# B&R Automation Studio project FeederLib
Automation Studio 4.10.2.37; technology packages: Acp10Arnc0 5.12.2, mapp 5.12.1, mappSafety 5.12.2, mappView 5.12.1

## Configuration Config1

CPU PC_any, AutomationRuntime C4.90, Build 4.1.2, Safety 0.0, Vc V4.72.2

### Task classes (Cpu.sw)
```
Cyclic#1 (cycle 2000 us, tolerance 200000 us):
  ReadData <- ReadData.prg
Cyclic#3 (cycle 100000 us):
  ReadTest <- ReadTest.prg
Binaries: mvLoader, udbdef, TCData, FWRules, arconfig, User, Role, iomap, asfw, ashwac, ashwd, sysconf, OpcUaMap
Libraries: sys_lib, AsBrStr, runtime, FeederLib, FileIO, standard, astime, arssl, asieccon
```

### Hardware
```
PC : PC_any v1.1.1.0 (OrderNumber=PC)
  ConfigurationID = FeederLib_Config1
  SystemTick = 2000
  IdleTaskClass = 4
  ActivateExceptionTaskClass = 1
  Cyclic1Duration = 2000
  Cyclic1Tolerance = 200000
  Cyclic2Duration = 50000
  Cyclic3Duration = 100000
  FileDevice1
  FileDeviceName1 = HardDisk
  FileDevicePath1 = D:\Users\stankevich.sl\Documents\FeederLib\Temp
  WebServerPort = 81
  ActivateOpcUa = 1
  OpcUaInformationModels_PV_Version = 1
```

## Configuration HW

CPU 5APC3100.KBU1-000, AutomationRuntime C4.90, Build 4.1.2, Safety 0.0, Vc V4.52.0

### Task classes (Cpu.sw)
```
Cyclic#1 (cycle 2000 us, tolerance 0 us):
  HWtest <- HWtest.prg
DataObjects: Acp10sys, assl1
NcDataObjects: acp10etxen <- acp10etxen.dob, gAxis01a <- gAxis01obj.gAxis01a.dob, gAxis01i <- gAxis01obj.gAxis01i.dob, gAxis02a <- gAxis02obj.gAxis02a.dob, gAxis02i <- gAxis02obj.gAxis02i.dob, acp10etxe1 <- acp10etxen.dob, gAxis02a1 <- gAxis02obj.gAxis02a.dob, gAxis02i1 <- gAxis02obj.gAxis02i.dob, gAxis01a1 <- gAxis01obj.gAxis01a.dob, gAxis01i1 <- gAxis01obj.gAxis01i.dob
Binaries: arsvcreg, udbdef, mvLoader, TCData, arflatprv, arcoal, Acp10map, acp10cfg, asnxdb1, Config_1, ashwd, ashwac, User, sysconf, asfw, arconfig, iomap, Role, Config, Settings, TCLang, Config_4, Config_2, Config_3, Config_7, Config_5, Config_6, Config_9, Config_8, asiol2, OpcUaMap, asiol1, AlarmCfg, AlarmHCfg, asnxdb2
Libraries: MpAxis, MpBase, NcGlobal, Acp10_MC, brsystem, Acp10man, sys_lib, Acp10par, runtime, FileIO, standard, astime, MpCom, AsBrStr, SfDomain, UserLib, asieccon, powerlnk, aruser, SfDomDrv, asusb, MpSfDomMgr, SfDomVis, arssl, asiodiag, astcp, dataobj, areventlog, UsAlarmLib, MpAlarmX, FeederLib
```

### Hardware
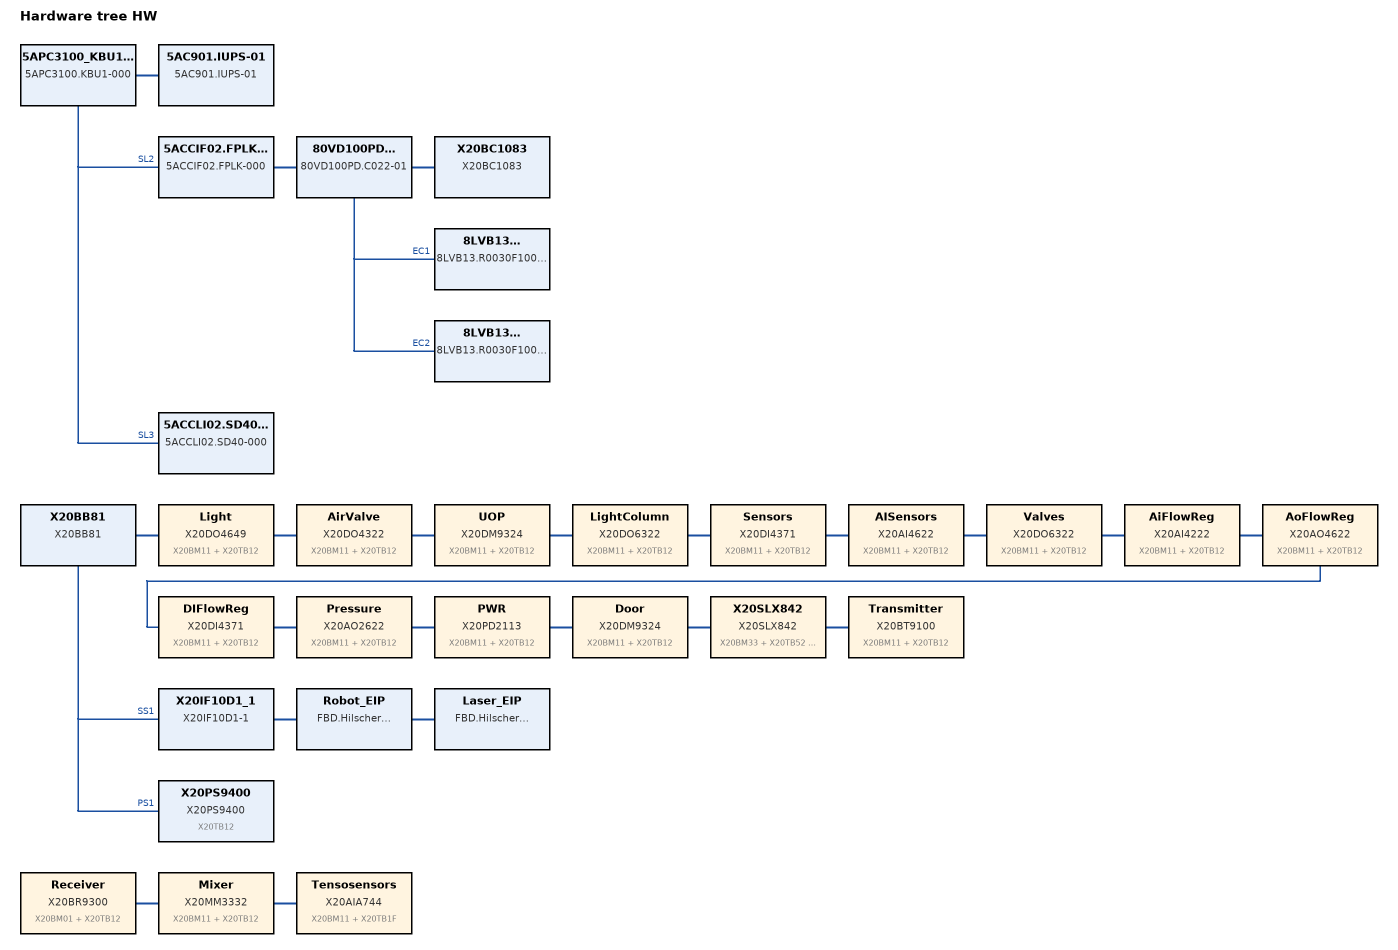
```
5AC901.IUPS-01 : 5AC901.IUPS-01 v1.3.1.0  [SL -> 5APC3100_KBU1_000.SL1]
5ACCIF02.FPLK-000 : 5ACCIF02.FPLK-000 v1.5.2.0  [SL -> 5APC3100_KBU1_000.SL2]
  Connector IF1:
    Channel1
    ChannelID1 = ACP10_MC_BROADCAST
    ChannelType1 = OCTET[24]
5ACCLI02.SD40-000 : 5ACCLI02.SD40-000 v2.0.0.0  [SL -> 5APC3100_KBU1_000.SL3]
5APC3100_KBU1_000 : 5APC3100.KBU1-000 v2.2.1.0
  Connector IF3:
    AssignedOperatingSystem = GPOS
  Connector IF4:
    AssignedOperatingSystem = ARemb
    ActivateDevice = 1
    Mode = Manual
    InternetAddress = 192.168.1.3
    SubnetMask = 255.255.255.0
  Connector IF9:
    OperatingSystem = ARemb
    ActivateDevice = 1
  Connector IF5:
    AssignedOperatingSystem = GPOS
  Connector IF6:
    AssignedOperatingSystem = GPOS
  Connector IF7:
    AssignedOperatingSystem = ARemb
  Connector IF8:
    AssignedOperatingSystem = ARemb
  ConfigurationID = 5in1
  ConfigVersion = 2.0.0
  UserPartitionSize = 100
  UserRamDevice = PCI.2.FPLK.SRAM
  UserRamSize = 520000
  RemMemDevice = PCI.2.FPLK.SRAM
  RemMemSize = 100000
  PermanentPvSize = 50
  RemanentGlobalPvSize = 1200
  EnableUsbRemoteInstall = 1
  EnableCfRemoteInstall = 1
  RebootReset = 1
  TimerDeviceType = EPLX2X
  TimerDevice = 5ACCIF02.FPLK-000.IF1
  TaskClassIdleTime = 2000
  Cyclic1Duration = 2000
  Cyclic1Tolerance = 0
  Cyclic2Tolerance = 0
  Cyclic3Tolerance = 0
  FileDevice1
  FileDeviceName1 = UserDev
  FileDevicePath1 = F:\
  FileDevice2
  FileDeviceName2 = Settings
  FileDevicePath2 = F:\Settings
  FtpUser1
  FtpUsername1 = service
  FtpUserPassword1 = FnTu9SDAOUjHE2rhZgIyHa2NFgHYN5XeFFIYZLvRcYw=
  FtpUserSalt1 = Afegl0l4
  FTPAccessRight1 = 0
  WebServerPort = 81
  ActivateOpcUa = 1
  OpcUaInformationModels_PV_Version = 1
  ActivateHypervisor = 1
80VD100PD.C022-01 : 80VD100PD.C022-01 v2.5.0.0  [PLK1 -> 5ACCIF02.FPLK-000.IF1 (NodeNumber=2) [Cable Type=PowerlinkCable, Length=10, Version=1.0.0.3]; PLK2 -> X20BC1083.PLK1 (NodeNumber=2) [Cable Type=PowerlinkCable, Length=10, Version=1.0.0.3]; EC1 -> 8LVB13.R0030F100-0.EC; EC2 -> 8LVB13.R0030F100-0a.EC; MT2 -> 8LVB13.R0030F100-0a.MT]
  MotionTP = Acp10Arnc0
  AxisIsPeriodic_r1 = on
  QuickStopIsNormallyOpen_r1 = on
  AxisIsPeriodic_r2 = on
  QuickStopIsNormallyOpen_r2 = on
8LVB13.R0030F100-0 : 8LVB13.R0030F100-0 v2.2.0.3  [EC -> 80VD100PD.C022-01.EC1; MT -> 80VD100PD.C022-01.MT1]
8LVB13.R0030F100-0a : 8LVB13.R0030F100-0 v2.2.0.3  [EC -> 80VD100PD.C022-01.EC2; MT -> 80VD100PD.C022-01.MT2]
AISensors : X20AI4622 v1.1.0.0  [SS1 -> X20TB12f.SS; SL -> X20BM11f.SL1]
  InputFilter = level 128
  ChannelType01 = 4 to 20mA
  ChannelType02 = 4 to 20mA
  ChannelType03 = 4 to 20mA
AiFlowReg : X20AI4222 v1.1.0.0  [SS1 -> X20TB12h.SS; SL -> X20BM11h.SL1]
AirValve : X20DO4322 v1.1.0.0  [SS1 -> X20TB12b.SS; SL -> X20BM11b.SL1]
AoFlowReg : X20AO4622 v1.2.0.0  [SS1 -> X20TB12j.SS; SL -> X20BM11j.SL1]
DIFlowReg : X20DI4371 v1.1.0.0  [SS1 -> X20TB12k.SS; SL -> X20BM11k.SL1]
Door : X20DM9324 v1.1.0.0  [SS1 -> X20TB12.SS; SL -> X20BM11.SL1]
Laser_EIP : FBD.Hilscher.EIGAdapterDTM.ENIP Generic Adapter v1.1100.6.6839 (OrderNumber=ENIP Generic Adapter, VendorAddress=192.168.10.1)  [EIP1 -> Robot_EIP.EIP2]
  DtmId = 5db86292-2f64-4b3a-8f97-36f326a2392b
  ChannelBlocks_1ab36399-b97a-45c0-9e04-50eb06144ae9  // Module 0
  IO_InputImage_1ab36399-b97a-45c0-9e04-50eb06144ae9  // 2 Byte(s)
  Channel_1_IO_InputImage_1ab36399-b97a-45c0-9e04-50eb06144ae9
  Name_Channel_1_IO_InputImage_1ab36399-b97a-45c0-9e04-50eb06144ae9 = Laser_is_assigned
  Channel_2_IO_InputImage_1ab36399-b97a-45c0-9e04-50eb06144ae9
  Name_Channel_2_IO_InputImage_1ab36399-b97a-45c0-9e04-50eb06144ae9 = Laser_is_ON
  Channel_3_IO_InputImage_1ab36399-b97a-45c0-9e04-50eb06144ae9
  Name_Channel_3_IO_InputImage_1ab36399-b97a-45c0-9e04-50eb06144ae9 = System_error
  Channel_4_IO_InputImage_1ab36399-b97a-45c0-9e04-50eb06144ae9
  Name_Channel_4_IO_InputImage_1ab36399-b97a-45c0-9e04-50eb06144ae9 = Guide_laser_is_ON
  Channel_5_IO_InputImage_1ab36399-b97a-45c0-9e04-50eb06144ae9
  Name_Channel_5_IO_InputImage_1ab36399-b97a-45c0-9e04-50eb06144ae9 = Program_active
  Channel_6_IO_InputImage_1ab36399-b97a-45c0-9e04-50eb06144ae9
  Name_Channel_6_IO_InputImage_1ab36399-b97a-45c0-9e04-50eb06144ae9 = End_of_program
  Channel_7_IO_InputImage_1ab36399-b97a-45c0-9e04-50eb06144ae9
  Name_Channel_7_IO_InputImage_1ab36399-b97a-45c0-9e04-50eb06144ae9 = Program_is_interrupted
  Channel_8_IO_InputImage_1ab36399-b97a-45c0-9e04-50eb06144ae9
  Name_Channel_8_IO_InputImage_1ab36399-b97a-45c0-9e04-50eb06144ae9 = Analog_control_is_ON
  Channel_9_IO_InputImage_1ab36399-b97a-45c0-9e04-50eb06144ae9
  Name_Channel_9_IO_InputImage_1ab36399-b97a-45c0-9e04-50eb06144ae9 = System_warning
  Channel_10_IO_InputImage_1ab36399-b97a-45c0-9e04-50eb06144ae9
  Name_Channel_10_IO_InputImage_1ab36399-b97a-45c0-9e04-50eb06144ae9 = Laser_is_ready
  Channel_11_IO_InputImage_1ab36399-b97a-45c0-9e04-50eb06144ae9
  Name_Channel_11_IO_InputImage_1ab36399-b97a-45c0-9e04-50eb06144ae9 = Emission_is_ON
  Channel_12_IO_InputImage_1ab36399-b97a-45c0-9e04-50eb06144ae9
  Name_Channel_12_IO_InputImage_1ab36399-b97a-45c0-9e04-50eb06144ae9 = Synchronization_output
  Channel_13_IO_InputImage_1ab36399-b97a-45c0-9e04-50eb06144ae9
  Name_Channel_13_IO_InputImage_1ab36399-b97a-45c0-9e04-50eb06144ae9 = Robot_mode
  Channel_14_IO_InputImage_1ab36399-b97a-45c0-9e04-50eb06144ae9
  Name_Channel_14_IO_InputImage_1ab36399-b97a-45c0-9e04-50eb06144ae9 = Interlock
  Channel_15_IO_InputImage_1ab36399-b97a-45c0-9e04-50eb06144ae9
  Name_Channel_15_IO_InputImage_1ab36399-b97a-45c0-9e04-50eb06144ae9 = Laser_alive
  Channel_16_IO_InputImage_1ab36399-b97a-45c0-9e04-50eb06144ae9
  Name_Channel_16_IO_InputImage_1ab36399-b97a-45c0-9e04-50eb06144ae9 = Ext_software_control_is_active
  Channel_17_IO_InputImage_1ab36399-b97a-45c0-9e04-50eb06144ae9
  Name_Channel_17_IO_InputImage_1ab36399-b97a-45c0-9e04-50eb06144ae9 = Output_power
  Type_Channel_17_IO_InputImage_1ab36399-b97a-45c0-9e04-50eb06144ae9 = UINT
  Channel_18_IO_InputImage_1ab36399-b97a-45c0-9e04-50eb06144ae9
  Name_Channel_18_IO_InputImage_1ab36399-b97a-45c0-9e04-50eb06144ae9 = Optical_channel
  Type_Channel_18_IO_InputImage_1ab36399-b97a-45c0-9e04-50eb06144ae9 = USINT
  Channel_19_IO_InputImage_1ab36399-b97a-45c0-9e04-50eb06144ae9
  Name_Channel_19_IO_InputImage_1ab36399-b97a-45c0-9e04-50eb06144ae9 = Program_number
  Type_Channel_19_IO_InputImage_1ab36399-b97a-45c0-9e04-50eb06144ae9 = USINT
  Channel_20_IO_InputImage_1ab36399-b97a-45c0-9e04-50eb06144ae9
  Name_Channel_20_IO_InputImage_1ab36399-b97a-45c0-9e04-50eb06144ae9 = Laser_error
  Channel_21_IO_InputImage_1ab36399-b97a-45c0-9e04-50eb06144ae9
  Name_Channel_21_IO_InputImage_1ab36399-b97a-45c0-9e04-50eb06144ae9 = Laser_warning
  Channel_22_IO_InputImage_1ab36399-b97a-45c0-9e04-50eb06144ae9
  Name_Channel_22_IO_InputImage_1ab36399-b97a-45c0-9e04-50eb06144ae9 = Chiller_error
  Channel_23_IO_InputImage_1ab36399-b97a-45c0-9e04-50eb06144ae9
  Name_Channel_23_IO_InputImage_1ab36399-b97a-45c0-9e04-50eb06144ae9 = Chiller_warning
  Channel_24_IO_InputImage_1ab36399-b97a-45c0-9e04-50eb06144ae9
  Name_Channel_24_IO_InputImage_1ab36399-b97a-45c0-9e04-50eb06144ae9 = Safety_open
  Channel_25_IO_InputImage_1ab36399-b97a-45c0-9e04-50eb06144ae9
  Name_Channel_25_IO_InputImage_1ab36399-b97a-45c0-9e04-50eb06144ae9 = Channel_error
  Channel_26_IO_InputImage_1ab36399-b97a-45c0-9e04-50eb06144ae9
  Name_Channel_26_IO_InputImage_1ab36399-b97a-45c0-9e04-50eb06144ae9 = Laser_is_busy
  Channel_27_IO_InputImage_1ab36399-b97a-45c0-9e04-50eb06144ae9
  Name_Channel_27_IO_InputImage_1ab36399-b97a-45c0-9e04-50eb06144ae9 = Slot_error
  Channel_28_IO_InputImage_1ab36399-b97a-45c0-9e04-50eb06144ae9
  Name_Channel_28_IO_InputImage_1ab36399-b97a-45c0-9e04-50eb06144ae9 = Cabinet_door_open
  Channel_29_IO_InputImage_1ab36399-b97a-45c0-9e04-50eb06144ae9
  Name_Channel_29_IO_InputImage_1ab36399-b97a-45c0-9e04-50eb06144ae9 = Reserved_module_is_active
  Channel_30_IO_InputImage_1ab36399-b97a-45c0-9e04-50eb06144ae9
  Name_Channel_30_IO_InputImage_1ab36399-b97a-45c0-9e04-50eb06144ae9 = Reduced_active_modules
  Channel_31_IO_InputImage_1ab36399-b97a-45c0-9e04-50eb06144ae9
  Name_Channel_31_IO_InputImage_1ab36399-b97a-45c0-9e04-50eb06144ae9 = Reserved1
  Channel_32_IO_InputImage_1ab36399-b97a-45c0-9e04-50eb06144ae9
  Name_Channel_32_IO_InputImage_1ab36399-b97a-45c0-9e04-50eb06144ae9 = Module_power_supply_warning
  Channel_33_IO_InputImage_1ab36399-b97a-45c0-9e04-50eb06144ae9
  Name_Channel_33_IO_InputImage_1ab36399-b97a-45c0-9e04-50eb06144ae9 = Reserved2
  Channel_34_IO_InputImage_1ab36399-b97a-45c0-9e04-50eb06144ae9
  Name_Channel_34_IO_InputImage_1ab36399-b97a-45c0-9e04-50eb06144ae9 = Reserved3
  Channel_35_IO_InputImage_1ab36399-b97a-45c0-9e04-50eb06144ae9
  Name_Channel_35_IO_InputImage_1ab36399-b97a-45c0-9e04-50eb06144ae9 = Reserved4
  Channel_36_IO_InputImage_1ab36399-b97a-45c0-9e04-50eb06144ae9
  Name_Channel_36_IO_InputImage_1ab36399-b97a-45c0-9e04-50eb06144ae9 = Laser_number
  Type_Channel_36_IO_InputImage_1ab36399-b97a-45c0-9e04-50eb06144ae9 = USINT
  Channel_37_IO_InputImage_1ab36399-b97a-45c0-9e04-50eb06144ae9
  Name_Channel_37_IO_InputImage_1ab36399-b97a-45c0-9e04-50eb06144ae9 = Reserver5
  Type_Channel_37_IO_InputImage_1ab36399-b97a-45c0-9e04-50eb06144ae9 = USINT
  IO_OutputImage_1ab36399-b97a-45c0-9e04-50eb06144ae9  // 2 Byte(s)
  Channel_1_IO_OutputImage_1ab36399-b97a-45c0-9e04-50eb06144ae9
  Name_Channel_1_IO_OutputImage_1ab36399-b97a-45c0-9e04-50eb06144ae9 = Laser_request
  Channel_2_IO_OutputImage_1ab36399-b97a-45c0-9e04-50eb06144ae9
  Name_Channel_2_IO_OutputImage_1ab36399-b97a-45c0-9e04-50eb06144ae9 = Laser_ON
  Channel_3_IO_OutputImage_1ab36399-b97a-45c0-9e04-50eb06144ae9
  Name_Channel_3_IO_OutputImage_1ab36399-b97a-45c0-9e04-50eb06144ae9 = Reset_errors
  Channel_4_IO_OutputImage_1ab36399-b97a-45c0-9e04-50eb06144ae9
  Name_Channel_4_IO_OutputImage_1ab36399-b97a-45c0-9e04-50eb06144ae9 = Guide_laser_ON
  Channel_5_IO_OutputImage_1ab36399-b97a-45c0-9e04-50eb06144ae9
  Name_Channel_5_IO_OutputImage_1ab36399-b97a-45c0-9e04-50eb06144ae9 = Program_start
  Channel_6_IO_OutputImage_1ab36399-b97a-45c0-9e04-50eb06144ae9
  Name_Channel_6_IO_OutputImage_1ab36399-b97a-45c0-9e04-50eb06144ae9 = Program_stop
  Channel_7_IO_OutputImage_1ab36399-b97a-45c0-9e04-50eb06144ae9
  Name_Channel_7_IO_OutputImage_1ab36399-b97a-45c0-9e04-50eb06144ae9 = Reserved7
  Channel_8_IO_OutputImage_1ab36399-b97a-45c0-9e04-50eb06144ae9
  Name_Channel_8_IO_OutputImage_1ab36399-b97a-45c0-9e04-50eb06144ae9 = Analog_control_ON
  Channel_9_IO_OutputImage_1ab36399-b97a-45c0-9e04-50eb06144ae9
  Name_Channel_9_IO_OutputImage_1ab36399-b97a-45c0-9e04-50eb06144ae9 = Enable_ext_software_control
  Channel_10_IO_OutputImage_1ab36399-b97a-45c0-9e04-50eb06144ae9
  Name_Channel_10_IO_OutputImage_1ab36399-b97a-45c0-9e04-50eb06144ae9 = Set_ramp_up
  Channel_11_IO_OutputImage_1ab36399-b97a-45c0-9e04-50eb06144ae9
  Name_Channel_11_IO_OutputImage_1ab36399-b97a-45c0-9e04-50eb06144ae9 = Set_ramp_down
  Channel_12_IO_OutputImage_1ab36399-b97a-45c0-9e04-50eb06144ae9
  Name_Channel_12_IO_OutputImage_1ab36399-b97a-45c0-9e04-50eb06144ae9 = Synchronization_input
  Channel_13_IO_OutputImage_1ab36399-b97a-45c0-9e04-50eb06144ae9
  Name_Channel_13_IO_OutputImage_1ab36399-b97a-45c0-9e04-50eb06144ae9 = Reserved8
  Channel_14_IO_OutputImage_1ab36399-b97a-45c0-9e04-50eb06144ae9
  Name_Channel_14_IO_OutputImage_1ab36399-b97a-45c0-9e04-50eb06144ae9 = Reserved9
  Channel_15_IO_OutputImage_1ab36399-b97a-45c0-9e04-50eb06144ae9
  Name_Channel_15_IO_OutputImage_1ab36399-b97a-45c0-9e04-50eb06144ae9 = Reserved10
  Channel_16_IO_OutputImage_1ab36399-b97a-45c0-9e04-50eb06144ae9
  Name_Channel_16_IO_OutputImage_1ab36399-b97a-45c0-9e04-50eb06144ae9 = External_error
  Channel_17_IO_OutputImage_1ab36399-b97a-45c0-9e04-50eb06144ae9
  Name_Channel_17_IO_OutputImage_1ab36399-b97a-45c0-9e04-50eb06144ae9 = Power
  Type_Channel_17_IO_OutputImage_1ab36399-b97a-45c0-9e04-50eb06144ae9 = UINT
  Channel_18_IO_OutputImage_1ab36399-b97a-45c0-9e04-50eb06144ae9
  Name_Channel_18_IO_OutputImage_1ab36399-b97a-45c0-9e04-50eb06144ae9 = Optical_channel_
  Type_Channel_18_IO_OutputImage_1ab36399-b97a-45c0-9e04-50eb06144ae9 = USINT
  Channel_19_IO_OutputImage_1ab36399-b97a-45c0-9e04-50eb06144ae9
  Name_Channel_19_IO_OutputImage_1ab36399-b97a-45c0-9e04-50eb06144ae9 = Program_number_
  Type_Channel_19_IO_OutputImage_1ab36399-b97a-45c0-9e04-50eb06144ae9 = USINT
  Channel_20_IO_OutputImage_1ab36399-b97a-45c0-9e04-50eb06144ae9
  Name_Channel_20_IO_OutputImage_1ab36399-b97a-45c0-9e04-50eb06144ae9 = Ramping_time
  Type_Channel_20_IO_OutputImage_1ab36399-b97a-45c0-9e04-50eb06144ae9 = UINT
  Channel_21_IO_OutputImage_1ab36399-b97a-45c0-9e04-50eb06144ae9
  Name_Channel_21_IO_OutputImage_1ab36399-b97a-45c0-9e04-50eb06144ae9 = Laser_number_
  Type_Channel_21_IO_OutputImage_1ab36399-b97a-45c0-9e04-50eb06144ae9 = USINT
  Channel_22_IO_OutputImage_1ab36399-b97a-45c0-9e04-50eb06144ae9
  Name_Channel_22_IO_OutputImage_1ab36399-b97a-45c0-9e04-50eb06144ae9 = Reserved6
  Type_Channel_22_IO_OutputImage_1ab36399-b97a-45c0-9e04-50eb06144ae9 = USINT
Light : X20DO4649 v1.1.0.0  [SS1 -> X20TB12a.SS; SL -> X20BM11a.SL1]
LightColumn : X20DO6322 v1.1.0.0  [SS1 -> X20TB12d.SS; SL -> X20BM11d.SL1]
Mixer : X20MM3332 v1.1.0.0  [SS1 -> X20TB12p.SS; SL -> X20BM11o.SL1]
PWR : X20PD2113 v1.1.0.0  [SS1 -> X20TB12m.SS; SL -> X20BM11m.SL1]
Pressure : X20AO2622 v1.2.0.0  [SS1 -> X20TB12l.SS; SL -> X20BM11l.SL1]
Receiver : X20BR9300 v1.1.0.0  [SS1 -> X20TB12o.SS; SL -> X20BM01a.SL1; X2X1 -> Transmitter.X2X1 [Cable Type=X2XCable, Length=10, Version=1.0.0.3]]
Robot_EIP : FBD.Hilscher.EIGAdapterDTM.ENIP Generic Adapter v1.1100.6.6839 (OrderNumber=ENIP Generic Adapter, VendorAddress=192.168.10.2)  [EIP1 -> X20IF10D1_1.IF1]
  DtmId = aba9a34a-c52a-40cf-8487-2c047c18b069
  ChannelBlocks_9f1ee490-7d39-4fa2-ab93-255e4565e3a3  // Module 0
  IO_InputImage_9f1ee490-7d39-4fa2-ab93-255e4565e3a3  // 2 Byte(s)
  Channel_1_IO_InputImage_9f1ee490-7d39-4fa2-ab93-255e4565e3a3
  Name_Channel_1_IO_InputImage_9f1ee490-7d39-4fa2-ab93-255e4565e3a3 = Robot_DO_1
  Channel_2_IO_InputImage_9f1ee490-7d39-4fa2-ab93-255e4565e3a3
  Name_Channel_2_IO_InputImage_9f1ee490-7d39-4fa2-ab93-255e4565e3a3 = Robot_DO_2
  Channel_3_IO_InputImage_9f1ee490-7d39-4fa2-ab93-255e4565e3a3
  Name_Channel_3_IO_InputImage_9f1ee490-7d39-4fa2-ab93-255e4565e3a3 = Robot_DO_3
  Channel_4_IO_InputImage_9f1ee490-7d39-4fa2-ab93-255e4565e3a3
  Name_Channel_4_IO_InputImage_9f1ee490-7d39-4fa2-ab93-255e4565e3a3 = Robot_DO_4
  Channel_5_IO_InputImage_9f1ee490-7d39-4fa2-ab93-255e4565e3a3
  Name_Channel_5_IO_InputImage_9f1ee490-7d39-4fa2-ab93-255e4565e3a3 = Robot_DO_5
  Channel_6_IO_InputImage_9f1ee490-7d39-4fa2-ab93-255e4565e3a3
  Name_Channel_6_IO_InputImage_9f1ee490-7d39-4fa2-ab93-255e4565e3a3 = Robot_DO_6
  Channel_7_IO_InputImage_9f1ee490-7d39-4fa2-ab93-255e4565e3a3
  Name_Channel_7_IO_InputImage_9f1ee490-7d39-4fa2-ab93-255e4565e3a3 = Robot_DO_7
  Channel_8_IO_InputImage_9f1ee490-7d39-4fa2-ab93-255e4565e3a3
  Name_Channel_8_IO_InputImage_9f1ee490-7d39-4fa2-ab93-255e4565e3a3 = Robot_DO_8
  Channel_9_IO_InputImage_9f1ee490-7d39-4fa2-ab93-255e4565e3a3
  Name_Channel_9_IO_InputImage_9f1ee490-7d39-4fa2-ab93-255e4565e3a3 = Robot_DO_9
  Channel_10_IO_InputImage_9f1ee490-7d39-4fa2-ab93-255e4565e3a3
  Name_Channel_10_IO_InputImage_9f1ee490-7d39-4fa2-ab93-255e4565e3a3 = Robot_DO_10
  Channel_11_IO_InputImage_9f1ee490-7d39-4fa2-ab93-255e4565e3a3
  Name_Channel_11_IO_InputImage_9f1ee490-7d39-4fa2-ab93-255e4565e3a3 = Robot_DO_11
  Channel_12_IO_InputImage_9f1ee490-7d39-4fa2-ab93-255e4565e3a3
  Name_Channel_12_IO_InputImage_9f1ee490-7d39-4fa2-ab93-255e4565e3a3 = Robot_DO_12
  Channel_13_IO_InputImage_9f1ee490-7d39-4fa2-ab93-255e4565e3a3
  Name_Channel_13_IO_InputImage_9f1ee490-7d39-4fa2-ab93-255e4565e3a3 = Robot_DO_13
  Channel_14_IO_InputImage_9f1ee490-7d39-4fa2-ab93-255e4565e3a3
  Name_Channel_14_IO_InputImage_9f1ee490-7d39-4fa2-ab93-255e4565e3a3 = Robot_DO_14
  Channel_15_IO_InputImage_9f1ee490-7d39-4fa2-ab93-255e4565e3a3
  Name_Channel_15_IO_InputImage_9f1ee490-7d39-4fa2-ab93-255e4565e3a3 = Robot_DO_15
  Channel_16_IO_InputImage_9f1ee490-7d39-4fa2-ab93-255e4565e3a3
  Name_Channel_16_IO_InputImage_9f1ee490-7d39-4fa2-ab93-255e4565e3a3 = Robot_DO_16
  Channel_17_IO_InputImage_9f1ee490-7d39-4fa2-ab93-255e4565e3a3
  Name_Channel_17_IO_InputImage_9f1ee490-7d39-4fa2-ab93-255e4565e3a3 = Robot_DO_17
  Channel_18_IO_InputImage_9f1ee490-7d39-4fa2-ab93-255e4565e3a3
  Name_Channel_18_IO_InputImage_9f1ee490-7d39-4fa2-ab93-255e4565e3a3 = Robot_DO_18
  Channel_19_IO_InputImage_9f1ee490-7d39-4fa2-ab93-255e4565e3a3
  Name_Channel_19_IO_InputImage_9f1ee490-7d39-4fa2-ab93-255e4565e3a3 = Robot_DO_19
  Channel_20_IO_InputImage_9f1ee490-7d39-4fa2-ab93-255e4565e3a3
  Name_Channel_20_IO_InputImage_9f1ee490-7d39-4fa2-ab93-255e4565e3a3 = Robot_DO_20
  Channel_21_IO_InputImage_9f1ee490-7d39-4fa2-ab93-255e4565e3a3
  Name_Channel_21_IO_InputImage_9f1ee490-7d39-4fa2-ab93-255e4565e3a3 = Robot_DO_21
  Channel_22_IO_InputImage_9f1ee490-7d39-4fa2-ab93-255e4565e3a3
  Name_Channel_22_IO_InputImage_9f1ee490-7d39-4fa2-ab93-255e4565e3a3 = Robot_DO_22
  Channel_23_IO_InputImage_9f1ee490-7d39-4fa2-ab93-255e4565e3a3
  Name_Channel_23_IO_InputImage_9f1ee490-7d39-4fa2-ab93-255e4565e3a3 = Robot_DO_23
  Channel_24_IO_InputImage_9f1ee490-7d39-4fa2-ab93-255e4565e3a3
  Name_Channel_24_IO_InputImage_9f1ee490-7d39-4fa2-ab93-255e4565e3a3 = Robot_DO_24
  Channel_25_IO_InputImage_9f1ee490-7d39-4fa2-ab93-255e4565e3a3
  Name_Channel_25_IO_InputImage_9f1ee490-7d39-4fa2-ab93-255e4565e3a3 = Robot_DO_25
  Channel_26_IO_InputImage_9f1ee490-7d39-4fa2-ab93-255e4565e3a3
  Name_Channel_26_IO_InputImage_9f1ee490-7d39-4fa2-ab93-255e4565e3a3 = Robot_DO_26
  Channel_27_IO_InputImage_9f1ee490-7d39-4fa2-ab93-255e4565e3a3
  Name_Channel_27_IO_InputImage_9f1ee490-7d39-4fa2-ab93-255e4565e3a3 = Robot_DO_27
  Channel_28_IO_InputImage_9f1ee490-7d39-4fa2-ab93-255e4565e3a3
  Name_Channel_28_IO_InputImage_9f1ee490-7d39-4fa2-ab93-255e4565e3a3 = Robot_DO_28
  Channel_29_IO_InputImage_9f1ee490-7d39-4fa2-ab93-255e4565e3a3
  Name_Channel_29_IO_InputImage_9f1ee490-7d39-4fa2-ab93-255e4565e3a3 = Robot_DO_29
  Channel_30_IO_InputImage_9f1ee490-7d39-4fa2-ab93-255e4565e3a3
  Name_Channel_30_IO_InputImage_9f1ee490-7d39-4fa2-ab93-255e4565e3a3 = Robot_DO_30
  Channel_31_IO_InputImage_9f1ee490-7d39-4fa2-ab93-255e4565e3a3
  Name_Channel_31_IO_InputImage_9f1ee490-7d39-4fa2-ab93-255e4565e3a3 = Robot_DO_31
  Channel_32_IO_InputImage_9f1ee490-7d39-4fa2-ab93-255e4565e3a3
  Name_Channel_32_IO_InputImage_9f1ee490-7d39-4fa2-ab93-255e4565e3a3 = Robot_DO_32
  Channel_33_IO_InputImage_9f1ee490-7d39-4fa2-ab93-255e4565e3a3
  Name_Channel_33_IO_InputImage_9f1ee490-7d39-4fa2-ab93-255e4565e3a3 = Robot_DO_33
  Channel_34_IO_InputImage_9f1ee490-7d39-4fa2-ab93-255e4565e3a3
  Name_Channel_34_IO_InputImage_9f1ee490-7d39-4fa2-ab93-255e4565e3a3 = Robot_DO_34
  Channel_35_IO_InputImage_9f1ee490-7d39-4fa2-ab93-255e4565e3a3
  Name_Channel_35_IO_InputImage_9f1ee490-7d39-4fa2-ab93-255e4565e3a3 = Robot_DO_35
  Channel_36_IO_InputImage_9f1ee490-7d39-4fa2-ab93-255e4565e3a3
  Name_Channel_36_IO_InputImage_9f1ee490-7d39-4fa2-ab93-255e4565e3a3 = Robot_DO_36
  Channel_37_IO_InputImage_9f1ee490-7d39-4fa2-ab93-255e4565e3a3
  Name_Channel_37_IO_InputImage_9f1ee490-7d39-4fa2-ab93-255e4565e3a3 = Robot_DO_37
  Channel_38_IO_InputImage_9f1ee490-7d39-4fa2-ab93-255e4565e3a3
  Name_Channel_38_IO_InputImage_9f1ee490-7d39-4fa2-ab93-255e4565e3a3 = Robot_DO_38
  Channel_39_IO_InputImage_9f1ee490-7d39-4fa2-ab93-255e4565e3a3
  Name_Channel_39_IO_InputImage_9f1ee490-7d39-4fa2-ab93-255e4565e3a3 = Robot_DO_39
  Channel_40_IO_InputImage_9f1ee490-7d39-4fa2-ab93-255e4565e3a3
  Name_Channel_40_IO_InputImage_9f1ee490-7d39-4fa2-ab93-255e4565e3a3 = Robot_DO_40
  Channel_41_IO_InputImage_9f1ee490-7d39-4fa2-ab93-255e4565e3a3
  Name_Channel_41_IO_InputImage_9f1ee490-7d39-4fa2-ab93-255e4565e3a3 = Robot_DO_41
  Channel_42_IO_InputImage_9f1ee490-7d39-4fa2-ab93-255e4565e3a3
  Name_Channel_42_IO_InputImage_9f1ee490-7d39-4fa2-ab93-255e4565e3a3 = Robot_DO_42
  Channel_43_IO_InputImage_9f1ee490-7d39-4fa2-ab93-255e4565e3a3
  Name_Channel_43_IO_InputImage_9f1ee490-7d39-4fa2-ab93-255e4565e3a3 = Robot_DO_43
  Channel_44_IO_InputImage_9f1ee490-7d39-4fa2-ab93-255e4565e3a3
  Name_Channel_44_IO_InputImage_9f1ee490-7d39-4fa2-ab93-255e4565e3a3 = Robot_DO_44
  Channel_45_IO_InputImage_9f1ee490-7d39-4fa2-ab93-255e4565e3a3
  Name_Channel_45_IO_InputImage_9f1ee490-7d39-4fa2-ab93-255e4565e3a3 = Robot_DO_45
  Channel_46_IO_InputImage_9f1ee490-7d39-4fa2-ab93-255e4565e3a3
  Name_Channel_46_IO_InputImage_9f1ee490-7d39-4fa2-ab93-255e4565e3a3 = Robot_DO_46
  Channel_47_IO_InputImage_9f1ee490-7d39-4fa2-ab93-255e4565e3a3
  Name_Channel_47_IO_InputImage_9f1ee490-7d39-4fa2-ab93-255e4565e3a3 = Robot_DO_47
  Channel_48_IO_InputImage_9f1ee490-7d39-4fa2-ab93-255e4565e3a3
  Name_Channel_48_IO_InputImage_9f1ee490-7d39-4fa2-ab93-255e4565e3a3 = Robot_DO_48
  Channel_49_IO_InputImage_9f1ee490-7d39-4fa2-ab93-255e4565e3a3
  Name_Channel_49_IO_InputImage_9f1ee490-7d39-4fa2-ab93-255e4565e3a3 = Robot_DO_49
  Channel_50_IO_InputImage_9f1ee490-7d39-4fa2-ab93-255e4565e3a3
  Name_Channel_50_IO_InputImage_9f1ee490-7d39-4fa2-ab93-255e4565e3a3 = Robot_DO_50
  Channel_51_IO_InputImage_9f1ee490-7d39-4fa2-ab93-255e4565e3a3
  Name_Channel_51_IO_InputImage_9f1ee490-7d39-4fa2-ab93-255e4565e3a3 = Robot_DO_51
  Channel_52_IO_InputImage_9f1ee490-7d39-4fa2-ab93-255e4565e3a3
  Name_Channel_52_IO_InputImage_9f1ee490-7d39-4fa2-ab93-255e4565e3a3 = Robot_DO_52
  Channel_53_IO_InputImage_9f1ee490-7d39-4fa2-ab93-255e4565e3a3
  Name_Channel_53_IO_InputImage_9f1ee490-7d39-4fa2-ab93-255e4565e3a3 = Robot_DO_53
  Channel_54_IO_InputImage_9f1ee490-7d39-4fa2-ab93-255e4565e3a3
  Name_Channel_54_IO_InputImage_9f1ee490-7d39-4fa2-ab93-255e4565e3a3 = Robot_DO_54
  Channel_55_IO_InputImage_9f1ee490-7d39-4fa2-ab93-255e4565e3a3
  Name_Channel_55_IO_InputImage_9f1ee490-7d39-4fa2-ab93-255e4565e3a3 = Robot_DO_55
  Channel_56_IO_InputImage_9f1ee490-7d39-4fa2-ab93-255e4565e3a3
  Name_Channel_56_IO_InputImage_9f1ee490-7d39-4fa2-ab93-255e4565e3a3 = Robot_DO_56
  Channel_57_IO_InputImage_9f1ee490-7d39-4fa2-ab93-255e4565e3a3
  Name_Channel_57_IO_InputImage_9f1ee490-7d39-4fa2-ab93-255e4565e3a3 = Robot_DO_57
  Channel_58_IO_InputImage_9f1ee490-7d39-4fa2-ab93-255e4565e3a3
  Name_Channel_58_IO_InputImage_9f1ee490-7d39-4fa2-ab93-255e4565e3a3 = Robot_DO_58
  Channel_59_IO_InputImage_9f1ee490-7d39-4fa2-ab93-255e4565e3a3
  Name_Channel_59_IO_InputImage_9f1ee490-7d39-4fa2-ab93-255e4565e3a3 = Robot_DO_59
  Channel_60_IO_InputImage_9f1ee490-7d39-4fa2-ab93-255e4565e3a3
  Name_Channel_60_IO_InputImage_9f1ee490-7d39-4fa2-ab93-255e4565e3a3 = Robot_DO_60
  Channel_61_IO_InputImage_9f1ee490-7d39-4fa2-ab93-255e4565e3a3
  Name_Channel_61_IO_InputImage_9f1ee490-7d39-4fa2-ab93-255e4565e3a3 = Robot_DO_61
  Channel_62_IO_InputImage_9f1ee490-7d39-4fa2-ab93-255e4565e3a3
  Name_Channel_62_IO_InputImage_9f1ee490-7d39-4fa2-ab93-255e4565e3a3 = Robot_DO_62
  Channel_63_IO_InputImage_9f1ee490-7d39-4fa2-ab93-255e4565e3a3
  Name_Channel_63_IO_InputImage_9f1ee490-7d39-4fa2-ab93-255e4565e3a3 = Robot_DO_63
  Channel_64_IO_InputImage_9f1ee490-7d39-4fa2-ab93-255e4565e3a3
  Name_Channel_64_IO_InputImage_9f1ee490-7d39-4fa2-ab93-255e4565e3a3 = Robot_DO_64
  Channel_65_IO_InputImage_9f1ee490-7d39-4fa2-ab93-255e4565e3a3
  Name_Channel_65_IO_InputImage_9f1ee490-7d39-4fa2-ab93-255e4565e3a3 = Robot_GO_1
  Type_Channel_65_IO_InputImage_9f1ee490-7d39-4fa2-ab93-255e4565e3a3 = UINT
  Channel_66_IO_InputImage_9f1ee490-7d39-4fa2-ab93-255e4565e3a3
  Name_Channel_66_IO_InputImage_9f1ee490-7d39-4fa2-ab93-255e4565e3a3 = Robot_GO_2
  Type_Channel_66_IO_InputImage_9f1ee490-7d39-4fa2-ab93-255e4565e3a3 = UINT
  Channel_67_IO_InputImage_9f1ee490-7d39-4fa2-ab93-255e4565e3a3
  Name_Channel_67_IO_InputImage_9f1ee490-7d39-4fa2-ab93-255e4565e3a3 = Robot_GO_3
  Type_Channel_67_IO_InputImage_9f1ee490-7d39-4fa2-ab93-255e4565e3a3 = UINT
  Channel_68_IO_InputImage_9f1ee490-7d39-4fa2-ab93-255e4565e3a3
  Name_Channel_68_IO_InputImage_9f1ee490-7d39-4fa2-ab93-255e4565e3a3 = Robot_GO_4
  Type_Channel_68_IO_InputImage_9f1ee490-7d39-4fa2-ab93-255e4565e3a3 = UINT
  Channel_69_IO_InputImage_9f1ee490-7d39-4fa2-ab93-255e4565e3a3
  Name_Channel_69_IO_InputImage_9f1ee490-7d39-4fa2-ab93-255e4565e3a3 = Robot_GO_5
  Type_Channel_69_IO_InputImage_9f1ee490-7d39-4fa2-ab93-255e4565e3a3 = UINT
  Channel_70_IO_InputImage_9f1ee490-7d39-4fa2-ab93-255e4565e3a3
  Name_Channel_70_IO_InputImage_9f1ee490-7d39-4fa2-ab93-255e4565e3a3 = Robot_GO_6
  Type_Channel_70_IO_InputImage_9f1ee490-7d39-4fa2-ab93-255e4565e3a3 = UINT
  Channel_71_IO_InputImage_9f1ee490-7d39-4fa2-ab93-255e4565e3a3
  Name_Channel_71_IO_InputImage_9f1ee490-7d39-4fa2-ab93-255e4565e3a3 = Robot_GO_7
  Type_Channel_71_IO_InputImage_9f1ee490-7d39-4fa2-ab93-255e4565e3a3 = UINT
  Channel_72_IO_InputImage_9f1ee490-7d39-4fa2-ab93-255e4565e3a3
  Name_Channel_72_IO_InputImage_9f1ee490-7d39-4fa2-ab93-255e4565e3a3 = Robot_GO_8
  Type_Channel_72_IO_InputImage_9f1ee490-7d39-4fa2-ab93-255e4565e3a3 = UINT
  Channel_73_IO_InputImage_9f1ee490-7d39-4fa2-ab93-255e4565e3a3
  Name_Channel_73_IO_InputImage_9f1ee490-7d39-4fa2-ab93-255e4565e3a3 = Robot_GO_9
  Type_Channel_73_IO_InputImage_9f1ee490-7d39-4fa2-ab93-255e4565e3a3 = UINT
  Channel_74_IO_InputImage_9f1ee490-7d39-4fa2-ab93-255e4565e3a3
  Name_Channel_74_IO_InputImage_9f1ee490-7d39-4fa2-ab93-255e4565e3a3 = Robot_GO_10
  Type_Channel_74_IO_InputImage_9f1ee490-7d39-4fa2-ab93-255e4565e3a3 = UINT
  IO_OutputImage_9f1ee490-7d39-4fa2-ab93-255e4565e3a3  // 2 Byte(s)
  Channel_1_IO_OutputImage_9f1ee490-7d39-4fa2-ab93-255e4565e3a3
  Name_Channel_1_IO_OutputImage_9f1ee490-7d39-4fa2-ab93-255e4565e3a3 = Robot_DI_1
  Channel_2_IO_OutputImage_9f1ee490-7d39-4fa2-ab93-255e4565e3a3
  Name_Channel_2_IO_OutputImage_9f1ee490-7d39-4fa2-ab93-255e4565e3a3 = Robot_DI_2
  Channel_3_IO_OutputImage_9f1ee490-7d39-4fa2-ab93-255e4565e3a3
  Name_Channel_3_IO_OutputImage_9f1ee490-7d39-4fa2-ab93-255e4565e3a3 = Robot_DI_3
  Channel_4_IO_OutputImage_9f1ee490-7d39-4fa2-ab93-255e4565e3a3
  Name_Channel_4_IO_OutputImage_9f1ee490-7d39-4fa2-ab93-255e4565e3a3 = Robot_DI_4
  Channel_5_IO_OutputImage_9f1ee490-7d39-4fa2-ab93-255e4565e3a3
  Name_Channel_5_IO_OutputImage_9f1ee490-7d39-4fa2-ab93-255e4565e3a3 = Robot_DI_5
  Channel_6_IO_OutputImage_9f1ee490-7d39-4fa2-ab93-255e4565e3a3
  Name_Channel_6_IO_OutputImage_9f1ee490-7d39-4fa2-ab93-255e4565e3a3 = Robot_DI_6
  Channel_7_IO_OutputImage_9f1ee490-7d39-4fa2-ab93-255e4565e3a3
  Name_Channel_7_IO_OutputImage_9f1ee490-7d39-4fa2-ab93-255e4565e3a3 = Robot_DI_7
  Channel_8_IO_OutputImage_9f1ee490-7d39-4fa2-ab93-255e4565e3a3
  Name_Channel_8_IO_OutputImage_9f1ee490-7d39-4fa2-ab93-255e4565e3a3 = Robot_DI_8
  Channel_9_IO_OutputImage_9f1ee490-7d39-4fa2-ab93-255e4565e3a3
  Name_Channel_9_IO_OutputImage_9f1ee490-7d39-4fa2-ab93-255e4565e3a3 = Robot_DI_9
  Channel_10_IO_OutputImage_9f1ee490-7d39-4fa2-ab93-255e4565e3a3
  Name_Channel_10_IO_OutputImage_9f1ee490-7d39-4fa2-ab93-255e4565e3a3 = Robot_DI_10
  Channel_11_IO_OutputImage_9f1ee490-7d39-4fa2-ab93-255e4565e3a3
  Name_Channel_11_IO_OutputImage_9f1ee490-7d39-4fa2-ab93-255e4565e3a3 = Robot_DI_11
  Channel_12_IO_OutputImage_9f1ee490-7d39-4fa2-ab93-255e4565e3a3
  Name_Channel_12_IO_OutputImage_9f1ee490-7d39-4fa2-ab93-255e4565e3a3 = Robot_DI_12
  Channel_13_IO_OutputImage_9f1ee490-7d39-4fa2-ab93-255e4565e3a3
  Name_Channel_13_IO_OutputImage_9f1ee490-7d39-4fa2-ab93-255e4565e3a3 = Robot_DI_13
  Channel_14_IO_OutputImage_9f1ee490-7d39-4fa2-ab93-255e4565e3a3
  Name_Channel_14_IO_OutputImage_9f1ee490-7d39-4fa2-ab93-255e4565e3a3 = Robot_DI_14
  Channel_15_IO_OutputImage_9f1ee490-7d39-4fa2-ab93-255e4565e3a3
  Name_Channel_15_IO_OutputImage_9f1ee490-7d39-4fa2-ab93-255e4565e3a3 = Robot_DI_15
  Channel_16_IO_OutputImage_9f1ee490-7d39-4fa2-ab93-255e4565e3a3
  Name_Channel_16_IO_OutputImage_9f1ee490-7d39-4fa2-ab93-255e4565e3a3 = Robot_DI_16
  Channel_17_IO_OutputImage_9f1ee490-7d39-4fa2-ab93-255e4565e3a3
  Name_Channel_17_IO_OutputImage_9f1ee490-7d39-4fa2-ab93-255e4565e3a3 = Robot_DI_17
  Channel_18_IO_OutputImage_9f1ee490-7d39-4fa2-ab93-255e4565e3a3
  Name_Channel_18_IO_OutputImage_9f1ee490-7d39-4fa2-ab93-255e4565e3a3 = Robot_DI_18
  Channel_19_IO_OutputImage_9f1ee490-7d39-4fa2-ab93-255e4565e3a3
  Name_Channel_19_IO_OutputImage_9f1ee490-7d39-4fa2-ab93-255e4565e3a3 = Robot_DI_19
  Channel_20_IO_OutputImage_9f1ee490-7d39-4fa2-ab93-255e4565e3a3
  Name_Channel_20_IO_OutputImage_9f1ee490-7d39-4fa2-ab93-255e4565e3a3 = Robot_DI_20
  Channel_21_IO_OutputImage_9f1ee490-7d39-4fa2-ab93-255e4565e3a3
  Name_Channel_21_IO_OutputImage_9f1ee490-7d39-4fa2-ab93-255e4565e3a3 = Robot_DI_21
  Channel_22_IO_OutputImage_9f1ee490-7d39-4fa2-ab93-255e4565e3a3
  Name_Channel_22_IO_OutputImage_9f1ee490-7d39-4fa2-ab93-255e4565e3a3 = Robot_DI_22
  Channel_23_IO_OutputImage_9f1ee490-7d39-4fa2-ab93-255e4565e3a3
  Name_Channel_23_IO_OutputImage_9f1ee490-7d39-4fa2-ab93-255e4565e3a3 = Robot_DI_23
  Channel_24_IO_OutputImage_9f1ee490-7d39-4fa2-ab93-255e4565e3a3
  Name_Channel_24_IO_OutputImage_9f1ee490-7d39-4fa2-ab93-255e4565e3a3 = Robot_DI_24
  Channel_25_IO_OutputImage_9f1ee490-7d39-4fa2-ab93-255e4565e3a3
  Name_Channel_25_IO_OutputImage_9f1ee490-7d39-4fa2-ab93-255e4565e3a3 = Robot_DI_25
  Channel_26_IO_OutputImage_9f1ee490-7d39-4fa2-ab93-255e4565e3a3
  Name_Channel_26_IO_OutputImage_9f1ee490-7d39-4fa2-ab93-255e4565e3a3 = Robot_DI_26
  Channel_27_IO_OutputImage_9f1ee490-7d39-4fa2-ab93-255e4565e3a3
  Name_Channel_27_IO_OutputImage_9f1ee490-7d39-4fa2-ab93-255e4565e3a3 = Robot_DI_27
  Channel_28_IO_OutputImage_9f1ee490-7d39-4fa2-ab93-255e4565e3a3
  Name_Channel_28_IO_OutputImage_9f1ee490-7d39-4fa2-ab93-255e4565e3a3 = Robot_DI_28
  Channel_29_IO_OutputImage_9f1ee490-7d39-4fa2-ab93-255e4565e3a3
  Name_Channel_29_IO_OutputImage_9f1ee490-7d39-4fa2-ab93-255e4565e3a3 = Robot_DI_29
  Channel_30_IO_OutputImage_9f1ee490-7d39-4fa2-ab93-255e4565e3a3
  Name_Channel_30_IO_OutputImage_9f1ee490-7d39-4fa2-ab93-255e4565e3a3 = Robot_DI_30
  Channel_31_IO_OutputImage_9f1ee490-7d39-4fa2-ab93-255e4565e3a3
  Name_Channel_31_IO_OutputImage_9f1ee490-7d39-4fa2-ab93-255e4565e3a3 = Robot_DI_31
  Channel_32_IO_OutputImage_9f1ee490-7d39-4fa2-ab93-255e4565e3a3
  Name_Channel_32_IO_OutputImage_9f1ee490-7d39-4fa2-ab93-255e4565e3a3 = Robot_DI_32
  Channel_33_IO_OutputImage_9f1ee490-7d39-4fa2-ab93-255e4565e3a3
  Name_Channel_33_IO_OutputImage_9f1ee490-7d39-4fa2-ab93-255e4565e3a3 = Robot_DI_33
  Channel_34_IO_OutputImage_9f1ee490-7d39-4fa2-ab93-255e4565e3a3
  Name_Channel_34_IO_OutputImage_9f1ee490-7d39-4fa2-ab93-255e4565e3a3 = Robot_DI_34
  Channel_35_IO_OutputImage_9f1ee490-7d39-4fa2-ab93-255e4565e3a3
  Name_Channel_35_IO_OutputImage_9f1ee490-7d39-4fa2-ab93-255e4565e3a3 = Robot_DI_35
  Channel_36_IO_OutputImage_9f1ee490-7d39-4fa2-ab93-255e4565e3a3
  Name_Channel_36_IO_OutputImage_9f1ee490-7d39-4fa2-ab93-255e4565e3a3 = Robot_DI_36
  Channel_37_IO_OutputImage_9f1ee490-7d39-4fa2-ab93-255e4565e3a3
  Name_Channel_37_IO_OutputImage_9f1ee490-7d39-4fa2-ab93-255e4565e3a3 = Robot_DI_37
  Channel_38_IO_OutputImage_9f1ee490-7d39-4fa2-ab93-255e4565e3a3
  Name_Channel_38_IO_OutputImage_9f1ee490-7d39-4fa2-ab93-255e4565e3a3 = Robot_DI_38
  Channel_39_IO_OutputImage_9f1ee490-7d39-4fa2-ab93-255e4565e3a3
  Name_Channel_39_IO_OutputImage_9f1ee490-7d39-4fa2-ab93-255e4565e3a3 = Robot_DI_39
  Channel_40_IO_OutputImage_9f1ee490-7d39-4fa2-ab93-255e4565e3a3
  Name_Channel_40_IO_OutputImage_9f1ee490-7d39-4fa2-ab93-255e4565e3a3 = Robot_DI_40
  Channel_41_IO_OutputImage_9f1ee490-7d39-4fa2-ab93-255e4565e3a3
  Name_Channel_41_IO_OutputImage_9f1ee490-7d39-4fa2-ab93-255e4565e3a3 = Robot_DI_41
  Channel_42_IO_OutputImage_9f1ee490-7d39-4fa2-ab93-255e4565e3a3
  Name_Channel_42_IO_OutputImage_9f1ee490-7d39-4fa2-ab93-255e4565e3a3 = Robot_DI_42
  Channel_43_IO_OutputImage_9f1ee490-7d39-4fa2-ab93-255e4565e3a3
  Name_Channel_43_IO_OutputImage_9f1ee490-7d39-4fa2-ab93-255e4565e3a3 = Robot_DI_43
  Channel_44_IO_OutputImage_9f1ee490-7d39-4fa2-ab93-255e4565e3a3
  Name_Channel_44_IO_OutputImage_9f1ee490-7d39-4fa2-ab93-255e4565e3a3 = Robot_DI_44
  Channel_45_IO_OutputImage_9f1ee490-7d39-4fa2-ab93-255e4565e3a3
  Name_Channel_45_IO_OutputImage_9f1ee490-7d39-4fa2-ab93-255e4565e3a3 = Robot_DI_45
  Channel_46_IO_OutputImage_9f1ee490-7d39-4fa2-ab93-255e4565e3a3
  Name_Channel_46_IO_OutputImage_9f1ee490-7d39-4fa2-ab93-255e4565e3a3 = Robot_DI_46
  Channel_47_IO_OutputImage_9f1ee490-7d39-4fa2-ab93-255e4565e3a3
  Name_Channel_47_IO_OutputImage_9f1ee490-7d39-4fa2-ab93-255e4565e3a3 = Robot_DI_47
  Channel_48_IO_OutputImage_9f1ee490-7d39-4fa2-ab93-255e4565e3a3
  Name_Channel_48_IO_OutputImage_9f1ee490-7d39-4fa2-ab93-255e4565e3a3 = Robot_DI_48
  Channel_49_IO_OutputImage_9f1ee490-7d39-4fa2-ab93-255e4565e3a3
  Name_Channel_49_IO_OutputImage_9f1ee490-7d39-4fa2-ab93-255e4565e3a3 = Robot_DI_49
  Channel_50_IO_OutputImage_9f1ee490-7d39-4fa2-ab93-255e4565e3a3
  Name_Channel_50_IO_OutputImage_9f1ee490-7d39-4fa2-ab93-255e4565e3a3 = Robot_DI_50
  Channel_51_IO_OutputImage_9f1ee490-7d39-4fa2-ab93-255e4565e3a3
  Name_Channel_51_IO_OutputImage_9f1ee490-7d39-4fa2-ab93-255e4565e3a3 = Robot_DI_51
  Channel_52_IO_OutputImage_9f1ee490-7d39-4fa2-ab93-255e4565e3a3
  Name_Channel_52_IO_OutputImage_9f1ee490-7d39-4fa2-ab93-255e4565e3a3 = Robot_DI_52
  Channel_53_IO_OutputImage_9f1ee490-7d39-4fa2-ab93-255e4565e3a3
  Name_Channel_53_IO_OutputImage_9f1ee490-7d39-4fa2-ab93-255e4565e3a3 = Robot_DI_53
  Channel_54_IO_OutputImage_9f1ee490-7d39-4fa2-ab93-255e4565e3a3
  Name_Channel_54_IO_OutputImage_9f1ee490-7d39-4fa2-ab93-255e4565e3a3 = Robot_DI_54
  Channel_55_IO_OutputImage_9f1ee490-7d39-4fa2-ab93-255e4565e3a3
  Name_Channel_55_IO_OutputImage_9f1ee490-7d39-4fa2-ab93-255e4565e3a3 = Robot_DI_55
  Channel_56_IO_OutputImage_9f1ee490-7d39-4fa2-ab93-255e4565e3a3
  Name_Channel_56_IO_OutputImage_9f1ee490-7d39-4fa2-ab93-255e4565e3a3 = Robot_DI_56
  Channel_57_IO_OutputImage_9f1ee490-7d39-4fa2-ab93-255e4565e3a3
  Name_Channel_57_IO_OutputImage_9f1ee490-7d39-4fa2-ab93-255e4565e3a3 = Robot_DI_57
  Channel_58_IO_OutputImage_9f1ee490-7d39-4fa2-ab93-255e4565e3a3
  Name_Channel_58_IO_OutputImage_9f1ee490-7d39-4fa2-ab93-255e4565e3a3 = Robot_DI_58
  Channel_59_IO_OutputImage_9f1ee490-7d39-4fa2-ab93-255e4565e3a3
  Name_Channel_59_IO_OutputImage_9f1ee490-7d39-4fa2-ab93-255e4565e3a3 = Robot_DI_59
  Channel_60_IO_OutputImage_9f1ee490-7d39-4fa2-ab93-255e4565e3a3
  Name_Channel_60_IO_OutputImage_9f1ee490-7d39-4fa2-ab93-255e4565e3a3 = Robot_DI_60
  Channel_61_IO_OutputImage_9f1ee490-7d39-4fa2-ab93-255e4565e3a3
  Name_Channel_61_IO_OutputImage_9f1ee490-7d39-4fa2-ab93-255e4565e3a3 = Robot_DI_61
  Channel_62_IO_OutputImage_9f1ee490-7d39-4fa2-ab93-255e4565e3a3
  Name_Channel_62_IO_OutputImage_9f1ee490-7d39-4fa2-ab93-255e4565e3a3 = Robot_DI_62
  Channel_63_IO_OutputImage_9f1ee490-7d39-4fa2-ab93-255e4565e3a3
  Name_Channel_63_IO_OutputImage_9f1ee490-7d39-4fa2-ab93-255e4565e3a3 = Robot_DI_63
  Channel_64_IO_OutputImage_9f1ee490-7d39-4fa2-ab93-255e4565e3a3
  Name_Channel_64_IO_OutputImage_9f1ee490-7d39-4fa2-ab93-255e4565e3a3 = Robot_DI_64
  Channel_65_IO_OutputImage_9f1ee490-7d39-4fa2-ab93-255e4565e3a3
  Name_Channel_65_IO_OutputImage_9f1ee490-7d39-4fa2-ab93-255e4565e3a3 = Robot_GI_1
  Type_Channel_65_IO_OutputImage_9f1ee490-7d39-4fa2-ab93-255e4565e3a3 = UINT
  Channel_66_IO_OutputImage_9f1ee490-7d39-4fa2-ab93-255e4565e3a3
  Name_Channel_66_IO_OutputImage_9f1ee490-7d39-4fa2-ab93-255e4565e3a3 = Robot_GI_2
  Type_Channel_66_IO_OutputImage_9f1ee490-7d39-4fa2-ab93-255e4565e3a3 = UINT
  Channel_67_IO_OutputImage_9f1ee490-7d39-4fa2-ab93-255e4565e3a3
  Name_Channel_67_IO_OutputImage_9f1ee490-7d39-4fa2-ab93-255e4565e3a3 = Robot_GI_3
  Type_Channel_67_IO_OutputImage_9f1ee490-7d39-4fa2-ab93-255e4565e3a3 = UINT
  Channel_68_IO_OutputImage_9f1ee490-7d39-4fa2-ab93-255e4565e3a3
  Name_Channel_68_IO_OutputImage_9f1ee490-7d39-4fa2-ab93-255e4565e3a3 = Robot_GI_4
  Type_Channel_68_IO_OutputImage_9f1ee490-7d39-4fa2-ab93-255e4565e3a3 = UINT
Sensors : X20DI4371 v1.1.0.0  [SS1 -> X20TB12e.SS; SL -> X20BM11e.SL1]
Tensosensors : X20AIA744 v1.3.0.0  [SS1 -> X20TB1F1.SS; SL -> X20BM11p.SL1]
Transmitter : X20BT9100 v1.1.0.0  [SS1 -> X20TB12n.SS; SL -> X20BM11n.SL1]
UOP : X20DM9324 v1.1.0.0  [SS1 -> X20TB12c.SS; SL -> X20BM11c.SL1]
Valves : X20DO6322 v1.1.0.0  [SS1 -> X20TB12g.SS; SL -> X20BM11g.SL1]
X20BB81 : X20BB81 v1.0.2.0
X20BC1083 : X20BC1083 v2.12.0.0  [PLK1 -> 80VD100PD.C022-01.PLK2 (NodeNumber=3) [Cable Type=PowerlinkCable, Length=10, Version=1.0.0.3]; SL -> X20BB81.SL1]
X20BM01a : X20BM01 v2.1.0.0
X20BM11 : X20BM11 v1.0.0.1  [X2X1 -> X20BM11m.X2X2]
X20BM11a : X20BM11 v1.0.0.1  [X2X1 -> X20BB81.IF1]
X20BM11b : X20BM11 v1.0.0.1  [X2X1 -> X20BM11a.X2X2]
X20BM11c : X20BM11 v1.0.0.1  [X2X1 -> X20BM11b.X2X2]
X20BM11d : X20BM11 v1.0.0.1  [X2X1 -> X20BM11c.X2X2]
X20BM11e : X20BM11 v1.0.0.1  [X2X1 -> X20BM11d.X2X2]
X20BM11f : X20BM11 v1.0.0.1  [X2X1 -> X20BM11e.X2X2]
X20BM11g : X20BM11 v1.0.0.1  [X2X1 -> X20BM11f.X2X2]
X20BM11h : X20BM11 v1.0.0.1  [X2X1 -> X20BM11g.X2X2]
X20BM11j : X20BM11 v1.0.0.1  [X2X1 -> X20BM11h.X2X2]
X20BM11k : X20BM11 v1.0.0.1  [X2X1 -> X20BM11j.X2X2]
X20BM11l : X20BM11 v1.0.0.1  [X2X1 -> X20BM11k.X2X2]
X20BM11m : X20BM11 v1.0.0.1  [X2X1 -> X20BM11l.X2X2]
X20BM11n : X20BM11 v1.0.0.1  [X2X1 -> X20BM33.X2X2]
X20BM11o : X20BM11 v1.0.0.1  [X2X1 -> X20BM01a.X2X2]
X20BM11p : X20BM11 v1.0.0.1  [X2X1 -> X20BM11o.X2X2]
X20BM33 : X20BM33 v1.0.0.6  [X2X1 -> X20BM11.X2X2]
X20IF10D1_1 : X20IF10D1-1 v1.6.0.0  [SS -> X20BB81.SS1]
  Connector IF1:
    DtmId = 89c72c1d-13b9-4e5d-9bc0-35ee8e3ffdec
  ConfigFile = X20IF10D1_1.dtm
  ConfigModule = asnxdb1
  CycleTime = 2000
X20PS9400 : X20PS9400 v1.4.0.0  [SS1 -> X20TB12q.SS; PS -> X20BB81.PS1]
  PowerInfo = on
X20SLX842 : X20SLX842 v2.2.0.0  [SS1 -> X20TB52.SS; SS2 -> X20TB52a.SS; SL -> X20BM33.SL1]
  Supervision = off
  SafeProject = SafeLOGIC-1
  SafeDesigner = 4.4.0.0
  DigitalOutput01 = viaSafeLOGIC
  DigitalOutput02 = viaSafeLOGIC
  DigitalOutput03 = viaSafeLOGIC
  DigitalOutput04 = viaSafeLOGIC
  DigitalOutput05 = viaSafeLOGIC
  DigitalOutput06 = viaSafeLOGIC
X20TB12 : X20TB12 v1.0.0.0
X20TB12a : X20TB12 v1.0.0.0
X20TB12b : X20TB12 v1.0.0.0
X20TB12c : X20TB12 v1.0.0.0
X20TB12d : X20TB12 v1.0.0.0
X20TB12e : X20TB12 v1.0.0.0
X20TB12f : X20TB12 v1.0.0.0
X20TB12g : X20TB12 v1.0.0.0
X20TB12h : X20TB12 v1.0.0.0
X20TB12j : X20TB12 v1.0.0.0
X20TB12k : X20TB12 v1.0.0.0
X20TB12l : X20TB12 v1.0.0.0
X20TB12m : X20TB12 v1.0.0.0
X20TB12n : X20TB12 v1.0.0.0
X20TB12o : X20TB12 v1.0.0.0
X20TB12p : X20TB12 v1.0.0.0
X20TB12q : X20TB12 v1.0.0.0
X20TB1F1 : X20TB1F v1.0.0.0
X20TB52 : X20TB52 v1.0.0.2
X20TB52a : X20TB52 v1.0.0.2
```

### IoMap.iom - 5APC3100_KBU1_000/IoMap.iom
```iecst
VAR_CONFIG
	Cyclic#1.::HWtest:FeederBlock.IOout.PrimaryFeeder.doMixer AT %QX."Mixer".StartChannel01;
	Cyclic#1.::HWtest:FeederBlock.IOout.SecondaryFeeder.doMixer AT %QX."Mixer".StartChannel02;
	Cyclic#1.::HWtest:FeederBlock.IOin.PrimaryFeeder.aiWeight AT %ID."Tensosensors".AnalogInput01;
	Cyclic#1.::HWtest:FeederBlock.IOin.SecondaryFeeder.aiWeight AT %ID."Tensosensors".AnalogInput02;
	Cyclic#1.::HWtest:FeederBlock.Config.PrimaryFeeder.ControlWord AT %QW."Tensosensors".ControlPacked01;
	Cyclic#1.::HWtest:FeederBlock.Config.SecondaryFeeder.ControlWord AT %QW."Tensosensors".ControlPacked02;
	Cyclic#1.::gLaserIO.Out.doPowerSupply AT %IX."X20SLX842".BOOL001;
	Cyclic#1.gSealedChamberIO.Out.BasicChamberIOOut.doBlockDoor[0] AT %QX."X20SLX842".BOOL101;
	Cyclic#1.gSealedChamberIO.In.BasicChamberIOIn.diDoorState[0].DoorIsClosed AT %QX."X20SLX842".BOOL102;
	Cyclic#1.::HWtest:FeederBlock.IOout.PrimaryFeeder.doShutOff AT %QX."Valves".DigitalOutput01;
	Cyclic#1.::HWtest:FeederBlock.IOout.SecondaryFeeder.doShutOff AT %QX."Valves".DigitalOutput02;
	Cyclic#1.::HWtest:FeederBlock.Control.PrimaryStart AT %IX."Robot_EIP".Robot_DO_5;
	Cyclic#1.::HWtest:FeederBlock.Control.SecondaryStart AT %IX."Robot_EIP".Robot_DO_6;
	Cyclic#1.::HWtest:FeederBlock.Control.PrimaryFeeder.Handler.PowderRate AT %IW."Robot_EIP".Robot_GO_3;
	Cyclic#1.::HWtest:FeederBlock.Control.PrimaryFeeder.Handler.GasRate AT %IW."Robot_EIP".Robot_GO_4;
	Cyclic#1.::HWtest:FeederBlock.Control.SecondaryFeeder.Handler.PowderRate AT %IW."Robot_EIP".Robot_GO_5;
	Cyclic#1.::HWtest:FeederBlock.IOin.SecondaryFeeder.Handler.aiGasRate AT %IW."Robot_EIP".Robot_GO_6;
	Cyclic#1.::HWtest:FeederBlock.IOout.PrimaryFeeder.aoGasRate AT %QW."AoFlowReg".AnalogOutput02;
	Cyclic#1.::HWtest:FeederBlock.IOout.SecondaryFeeder.aoGasRate AT %QW."AoFlowReg".AnalogOutput03;
END_VAR
```

### Acp10cfg.ncc - 5APC3100_KBU1_000/Motion/Acp10cfg.ncc
```
NcConfiguration (Version=5.02.1, NcSwId=Acp10)
  ACP10CF1_typ:
    cnt_nettrc_rec_drive = 150
    bufsize_trace_upload = 1200
    tc_nc_man_task = Cyclic #1
    glob_pv_as_ncobject = Yes
    ncsys_dl_broadcast = Yes
    ncsys_dl_acp_reset = Yes
    safemc_log_err_to_ax = Yes
    network_init:
      ncsw_init_execute = Yes
      automatic_execute = No
      node_nr_warning = Yes
      net_err_before_ncact = Yes
    nettrc:
      enter_parsecrec = Yes
      enter_ncaction = Yes
      save_ring_startidx = No
    cam_prof_download:
      cam_dat_dl_parallel = No
      tc_cam_dl_parallel = Task class for NC Manager task
    plk_if[0]:
      if_name = IF3
      tc_CycDat_PLCopen = Task class for NC Manager task
      mc_broadcast_extdat = No
    plk_if[1]:
      if_name = SL2.IF1
      tc_CycDat_PLCopen = Task class for NC Manager task
      mc_broadcast_extdat = No
```

### Acp10map.ncm - 5APC3100_KBU1_000/Motion/Acp10map.ncm
```
NcMapping (NcSwId=Acp10)
  NcObject gAxis01 (ModuleId=80VD100PD.C022-01, Type=ncAXIS, Channel=1, AcoposSimulation=Off, InitParameter=gAxis01i, AcoposParameter=gAxis01a, AdditionalData=PLCopen_ModPos="1000,1" , Disabled=FALSE, ModuleDisabled=FALSE)
  NcObject gAxis02 (ModuleId=80VD100PD.C022-01, Type=ncAXIS, Channel=2, AcoposSimulation=Off, InitParameter=gAxis02i, AcoposParameter=gAxis02a, AdditionalData=PLCopen_ModPos="1000,1" , Disabled=FALSE, ModuleDisabled=FALSE)
  NcObject 80VD100PD.C022-01_ncV_AXIS1 (ModuleId=80VD100PD.C022-01, Type=ncV_AXIS, Channel=1, Disabled=TRUE, ModuleDisabled=FALSE)
  NcObject 80VD100PD.C022-01_ncV_AXIS2 (ModuleId=80VD100PD.C022-01, Type=ncV_AXIS, Channel=2, Disabled=TRUE, ModuleDisabled=FALSE)
```

### Config.mpaxisbasic - 5APC3100_KBU1_000/Motion/Config.mpaxisbasic
```
Element gLinkFeeder1 (Type=mpaxisbasic)
Element gLinkFeeder2 (Type=mpaxisbasic)
```

- Safety project (password-protected, skipped)

### Alarms.mpalarmxcore - 5APC3100_KBU1_000/mappServices/Alarms.mpalarmxcore
```
Element gAlarmXCore (Type=mpalarmxcore)
  mapp.AlarmX.Core:
    BySeverity:
      [0]:
        Severity = 1
        [0] = Reaction
          Name = ReactionWarning
      [1]:
        Severity = 5
        [0] = Reaction
          Name = ReactionWarningAlarm
      [2]:
        Severity = 9
        [0] = Reaction
          Name = ReactionAlarmStopAll
      [3]:
        Severity = 10
        [0] = Reaction
          Name = ReactionAlarmSignalAndStopAll
      [4]:
        Severity = 3
        [0] = Reaction
          Name = ReactionSignal
    Default:
      [0] = Reaction
```

## Logical view

Binary libraries used (declarations not repeated): operator, runtime, astime, AsIecCon, sys_lib, AsBrStr, FileIO, standard, MpAxis, Acp10_MC, NcGlobal, MpBase, MpCom, brsystem, Acp10man, Acp10par, SfDomain, MpAlarmX

### Global.var - Global variables
```iecst
VAR
	T : ARRAY[0..2399] OF REAL;
	Ktare : ARRAY[0..2399] OF REAL;
	V : ARRAY[0..2399] OF REAL;
	W : ARRAY[0..2399] OF REAL;
	gAxis02 : ACP10AXIS_typ;
	gAxis01 : ACP10AXIS_typ;
END_VAR
```

### Package Logical/Libraries - Global libraries

### Library Logical/Libraries/UserLib (IEC, version 1.01.0)

#### Types.typ - Exported data types
```iecst
(*----------------------------------------------------------------Others------------------------------------------------------------------------------------------------------------------------------------------*)

TYPE
	StepActiveEnumType :
		(
		STEPACTIVE_STOP,
		STEPACTIVE_INITIALIZATION,
		STEPACTIVE_RUN
		);
	Errors :
		(
		NO_ERRORS,
		ARGON_PRESSURE_IS_TO_LOW,
		AIR_PRESSURE_IS_TO_LOW
		);
	VentilateValveSensType : 	STRUCT
		TopVentilateValveIsOpened : BOOL;
		TopVentilateValveIsClosed : BOOL;
		BottomVentilateValveIsOpened : BOOL;
		BottomVentilateValveIsClosed : BOOL;
	END_STRUCT;
	CalibrationType : 	STRUCT
		A : REAL;
		B : REAL;
		C : REAL;
		MaxValue : REAL;
		MinValue : REAL;
	END_STRUCT;
	ReactionsType : 	STRUCT
		Warning : BOOL;
		WarningAlarm : BOOL;
		AlarmStopAll : BOOL;
		Signal : BOOL;
		AlarmSignalAndStopAll : BOOL;
	END_STRUCT;
	BlinkModeType :
		(
		BLINKMODE_CONSTANT_ON, (*Постоянный сигнал включен*)
		BLINKMODE_CONSTANT_OFF, (*Постоянный сигнал выключен*)
		BLINKMODE_SLOW, (*Мигание период 1000 мс*)
		BLINKMODE_MEDIUM, (*Мигание период 500 мс*)
		BLINKMODE_FAST (*Мигание период 250 мс*)
		);
	FBRobotAlarmsIOInType : 	STRUCT
		diRobotError : BOOL;
		diBatteryAlarm : BOOL;
		diESTOP : BOOL;
		diInputSimulated : BOOL;
		diOutputSimulated : BOOL;
	END_STRUCT;
END_TYPE

(*Sts*)

TYPE
	FBStatusEnumType :
		(
		Init := 0,
		Idle := 1,
		Bizy := 2,
		Done := 3,
		Error := 4
		);
END_TYPE
```

#### UserLib.fun - Exported functions and function blocks
```iecst
(*----------------------------------------------------------------Others------------------------------------------------------------------------------------------------------------------------------------------*)

{REDUND_OK} FUNCTION_BLOCK FBComparebValueDelay (*TODO: Add your comment here*) (*$GROUP=User,$CAT=User,$GROUPICON=User.png,$CATICON=User.png*)
	VAR_INPUT
		Delay : {REDUND_UNREPLICABLE} TIME; (*Задержка проверки переменной*)
		ActualValue : {REDUND_UNREPLICABLE} BOOL;
		TargetValue : {REDUND_UNREPLICABLE} BOOL;
	END_VAR
	VAR_OUTPUT
		Out : BOOL;
	END_VAR
	VAR
		TON_0 : TON;
		TON_1 : TON;
	END_VAR
END_FUNCTION_BLOCK

FUNCTION_BLOCK FBCountdownTimer
	VAR_INPUT
		Start : BOOL; (*Триггер на старт, пока он включен, таймер отсчитывает время*)
		Time : TIME; (*Заданное время до срабатывания таймера*)
	END_VAR
	VAR_OUTPUT
		TimeLeft : TIME; (*Актуальное время до срабатывания таймера*)
		DintTimeLeft : DINT; (*Актуальное время до срабатывания таймера*)
		StrTimeLeft : STRING[255]; (*Актуальное время до срабатывания таймера*)
		Stop : BOOL; (*Таймер закончил отсчет времени*)
	END_VAR
	VAR
		TON_0 : TON;
		temp_sec : DINT;
		temp_min : STRING[80];
		temp_str : STRING[80];
		zzEdge00000 : BOOL;
	END_VAR
END_FUNCTION_BLOCK

{REDUND_OK} FUNCTION InRange_Percent : BOOL (*TODO: Add your comment here*) (*$GROUP=User,$CAT=User,$GROUPICON=User.png,$CATICON=User.png*)
	VAR_INPUT
		ActualValue : REAL;
		TargetValue : REAL;
		DeviationInPercents : REAL; (*Значение несоответствия целевому в процентах*)
	END_VAR
	VAR
		DeviationValue : REAL;
		Value : REAL;
	END_VAR
END_FUNCTION

{REDUND_ERROR} FUNCTION CalibrateREAL : REAL (*Calibrate output signal by Ax2+Bx+C*) (*$GROUP=User,$CAT=User,$GROUPICON=User.png,$CATICON=User.png*)
	VAR_INPUT
		IN : REAL;
		CalibrationData : CalibrationType;
	END_VAR
	VAR
		value : REAL;
	END_VAR
END_FUNCTION

{REDUND_ERROR} FUNCTION Calibrate : INT (*Calibrate output signal by Ax2+Bx+C*) (*$GROUP=User,$CAT=User,$GROUPICON=User.png,$CATICON=User.png*)
	VAR_INPUT
		IN : INT;
		CalibrationData : CalibrationType;
	END_VAR
	VAR
		value : REAL;
	END_VAR
END_FUNCTION

{REDUND_OK} FUNCTION FBlink : BOOL (*TODO: Add your comment here*) (*$GROUP=User,$CAT=User,$GROUPICON=User.png,$CATICON=User.png*)
	VAR_INPUT
		BlinkMode : BlinkModeType;
	END_VAR
	VAR
		PulseTime : REAL;
		PauseTime : REAL;
		EnablePulse : BOOL;
	END_VAR
END_FUNCTION

{REDUND_OK} FUNCTION_BLOCK FBRobotAlarms (*TODO: Add your comment here*) (*$GROUP=User,$CAT=User,$GROUPICON=User.png,$CATICON=User.png*)
	VAR_INPUT
		IOIn : FBRobotAlarmsIOInType;
	END_VAR
	VAR
		(*AlarmsList : ARRAY[1..255] OF AlarmsListType := [(Name:='ErrorBatteryAlarm',Config:=(Code:=4000,Severity:=5)),254(0)];*)
		(*FBAlarmListDiscrValMon_0 : FBAlarmListDiscrValMon;*)
	END_VAR
END_FUNCTION_BLOCK
```

#### Calibrate.st
```iecst
(* Calibrate output signal by Ax2+Bx+C *)
FUNCTION Calibrate

	value := CalibrationData.A*IN*IN+CalibrationData.B*IN+CalibrationData.C;
	Calibrate := REAL_TO_INT(LIMIT(CalibrationData.MinValue, value, CalibrationData.MaxValue));

END_FUNCTION

(* Calibrate output signal by Ax2+Bx+C *)
FUNCTION CalibrateREAL

	value := CalibrationData.A*IN*IN+CalibrationData.B*IN+CalibrationData.C;
	CalibrateREAL := LIMIT(CalibrationData.MinValue, value, CalibrationData.MaxValue);

END_FUNCTION
```

#### Inrange_Percent.st
```iecst
FUNCTION InRange_Percent

	Value := ActualValue - TargetValue ;
	DeviationValue := TargetValue*(DeviationInPercents/100);

	IF (Value <= DeviationValue) AND (Value >= DeviationValue*(-1)) THEN
		InRange_Percent := TRUE ;
	END_IF

	IF (Value > DeviationValue) AND (Value < DeviationValue*(-1)) THEN
		InRange_Percent := FALSE ;
	END_IF

END_FUNCTION
```

#### FBComparebValueDelay.st
```iecst
(**************************************************************
* Функциональный блок: FBComparebValueDelay
* Файл: FBComparebValueDelay.st
* Создан: 18.11.2020
***************************************************************
* Описание:
- Функциональный блок позволяет сравнить две переменные с
заданной задержкой во времени
Это может быть полезно для мониторинга ошибок состояния
к примеру, мы хотим проследить, открылась ли шиберная заслонка,
но она имеет некую инерцию и закрывается не мгновенно, для этого мы
отслеживаем ее состояние через некоторый момент времени заданный
на входе в функциональный блок.

* Интерфейс
Входы:

- Delay (TIME) - задержка проверки переменной
- ActualValue (BOOL) - Текущее состояние
- TargetValue (BOOL) - Целевое состояние

Выход:
- Out (BOOL) - Если значения текущего состояния и целевого состояния
через delay времени равны между собой, то TRUE

***************************************************************
Версия  |     Дата     |    Автор     |         Описание
---------------------------------------------------------------
V1.00.0 | 18.11.2020   | Топалов И.К. | Написание ФБ
**************************************************************)

FUNCTION_BLOCK FBComparebValueDelay

	TON_0(PT := Delay, IN := TargetValue);
	TON_1(PT := Delay, IN := NOT TargetValue);

	IF TON_0.Q OR TON_1.Q THEN
	Out := ActualValue = TargetValue;
	END_IF

END_FUNCTION_BLOCK
```

#### FBCountdownTimer.st
```iecst
(**************************************************************
* Функциональный блок: FBCountdownTimer
* Файл: FBCountdownTimer.st
* Создан: 19.11.2020
***************************************************************
* Описание:
- Функциональный блок выполняет роль обратного таймера
с функцией срабатывания и выводом оставшегося времени

* Интерфейс
Входы:
- Start (BOOL) - Триггер на старт, пока он включен, таймер отсчитывает время
- Time (TIME) - Заданное время до срабатывания таймера

Выходы:
- TimeLeft (TIME) - Актуальное время до срабатывания таймера
- DintTimeLeft (DINT) - Актуальное время до срабатывания таймера
- StrTimeLeft (STRING255) - Актуальное время до срабатывания таймера
- Stop (BOOL) - Таймер закончил отсчет времени

***************************************************************
Версия  |     Дата     |    Автор     |         Описание
---------------------------------------------------------------
V1.00.0 | 19.11.2020   | Топалов И.К. | Написание ФБ
**************************************************************)

FUNCTION_BLOCK FBCountdownTimer

	TON_0(PT:= Time);
	IF EDGEPOS(Start) THEN
		TON_0.IN := TRUE;
	END_IF

	IF (NOT Start) THEN
		TON_0.IN := FALSE;
		Stop := FALSE;
	END_IF

	IF (TON_0.Q) THEN
		TON_0.IN := FALSE;
		Stop := TRUE;
	END_IF

	temp_sec := TIME_TO_DINT(Time - TON_0.ET)/1000;
	temp_min := DINT_TO_STRING(temp_sec/60);
	temp_min := CONCAT(temp_min,':');
	temp_str := DINT_TO_STRING(temp_sec MOD 60);

	StrTimeLeft := CONCAT(temp_min,temp_str);
	DintTimeLeft := temp_sec;
	TimeLeft := Time - TON_0.ET;

END_FUNCTION_BLOCK
```

#### FBlink.st
```iecst
(* TODO: Add your comment here *)
FUNCTION FBlink

	//LCRPFM_0(enable := EnablePulse, x := 1, max_value := 1, min_value := 0, t_pulse := PulseTime, t_pause := PauseTime);

	CASE BlinkMode  OF

		BLINKMODE_CONSTANT_OFF:

			EnablePulse := FALSE;

		BLINKMODE_CONSTANT_ON:

			EnablePulse := TRUE;
			PulseTime := 1;
			PauseTime := 0;

		BLINKMODE_SLOW:

			EnablePulse := TRUE;
			PulseTime := 1;
			PauseTime := 1;

		BLINKMODE_MEDIUM:

			EnablePulse := TRUE;
			PulseTime := 0.5;
			PauseTime := 0.5;

		BLINKMODE_FAST:

			EnablePulse := TRUE;
			PulseTime := 0.25;
			PauseTime := 0.25;

	END_CASE

END_FUNCTION
```

#### DeviceTypes.typ - Exported data types
```iecst
(*----------------------------------------------------------------Robot----------------------------------------------------------------------------------------------------------------------*)

TYPE
	IORobotEthIpType : 	STRUCT
		In : IORobotEthIpInType;
		Out : IORobotEthIpOutType;
	END_STRUCT;
	IORobotEthIpInType : 	STRUCT
		diLaserOn : BOOL;
		diProgramStop : BOOL;
		diPilotOn : BOOL;
		diCoaxArgon : BOOL;
		diBulbStart : ARRAY[1..10]OF BOOL;
		diCrossjetOn : BOOL;
		diPiezoRegHead : BOOL;
		diLaserRequest : BOOL;
		diAnalyseOn : BOOL;
		diAnalyseOff : BOOL;
		diPowderSwitchOn : BOOL;
		diRobotError : BOOL;
		diReady : BOOL;
		diProgRun : BOOL;
		diModeAuto : BOOL;
		diModeT2 : BOOL;
		diModeT1 : BOOL;
		diBatteryAlarm : BOOL;
		diESTOP : BOOL;
		diInputSimulated : BOOL;
		diOutputSimulated : BOOL;
		diProgPaused : BOOL;
		diBusy : BOOL;
		diTpEnabled : BOOL;
		diHold : BOOL;
		aiLaserPower : UINT;
		aiCoaxialGasSetpoint : UINT;
		aiHeadGasSetpiont : UINT;
		aiBulbGasSetpoint : ARRAY[1..10]OF UINT;
		aiLaserProgram : UINT;
		aiWobblerProgramNumber : UINT;
		aiWobblerAmplitude : UINT;
		aiWobblerFriequency : UINT;
	END_STRUCT;
	IORobotEthIpOutType : 	STRUCT
		doStart : BOOL;
		doStop : BOOL;
		doResetError : BOOL;
		doMachineError : BOOL;
	END_STRUCT;
END_TYPE
```

#### FBRobotAlarms.st
```iecst
(* TODO: Add your comment here *)
FUNCTION_BLOCK FBRobotAlarms
	//Не подключены
//	IOIn.diESTOP
//	IOIn.diInputSimulated
//	IOIn.diOutputSimulated
//	IOIn.diRobotError

	// Мониторинг ошибок
//	FBAlarmListDiscrValMon_0(Ena := TRUE, AlarmsList := AlarmsList, QuantityAlarms := 1, DeviceName := 'Робот');

//	AlarmsList[1].Monitoring.Monitored_PV := IOIn.diBatteryAlarm;

END_FUNCTION_BLOCK
```

### Library Logical/Libraries/UsAlarmLib (IEC)
Depends on: UserLib, MpAlarmX

#### UsAlarmLib.fun - Exported functions and function blocks
```iecst
(*----------------------------------------------------------------Alarms------------------------------------------------------------------------------------------------------------------------------------------*)

FUNCTION_BLOCK FBRecordAlarmsInCore
	VAR_INPUT
		Enable : BOOL;
		AlarmBVMListAdr : UDINT; (*Ссылка на массив алармов*)
		ListSize : USINT; (*Количество элементов в массиве*)
		AlarmXCore : MpComIdentType;
		Prefix : STRING[80];
		DeviceName : STRING[80];
		ResetError : BOOL;
	END_VAR
	VAR_OUTPUT
		Status : AlarmControlStatusTypeEnum := AlarmControl_INIT;
	END_VAR
	VAR
		i : USINT := 0;
		MpAlarmXAlarmConfigType_0 : MpAlarmXAlarmConfigType;
		MpAlarmXConfigAlarm_0 : MpAlarmXConfigAlarm;
		AlarmBVMListItem : REFERENCE TO AlarmBVMItemType;
	END_VAR
END_FUNCTION_BLOCK

FUNCTION_BLOCK FBCheckAlarmValues
	VAR_INPUT
		Enable : BOOL;
		AlarmBVMListAdr : UDINT; (*Ссылка на массив алармов*)
		ListSize : USINT; (*Количество элементов в массиве*)
		AlarmXCore : MpComIdentType;
		ResetError : BOOL;
	END_VAR
	VAR_OUTPUT
		Status : AlarmControlStatusTypeEnum := AlarmControl_INIT;
	END_VAR
	VAR
		i : USINT := 0;
		AlarmListItem : REFERENCE TO AlarmBVMItemType;
		boolVal : REFERENCE TO BOOL; (*Value for compare monitoried and trigger values*)
		AlarmXSetStatus : DINT;
		AlarmXResetStatus : DINT;
	END_VAR
END_FUNCTION_BLOCK

{REDUND_ERROR} FUNCTION_BLOCK FBAlarmListControl (*TODO: Add your comment here*) (*$GROUP=User,$CAT=User,$GROUPICON=User.png,$CATICON=User.png*)
	VAR_INPUT
		Enable : BOOL;
		AlarmBVMListAdr : UDINT; (*Ссылка на массив алармов*)
		ListSize : USINT; (*Количество элементов в массиве*)
		AlarmXCore : MpComIdentType;
		Prefix : STRING[80];
		DeviceName : STRING[80];
		ResetError : BOOL;
	END_VAR
	VAR_OUTPUT
		Status : AlarmControlStatusTypeEnum := AlarmControl_INIT;
	END_VAR
	VAR
		RecordAlarm : FBRecordAlarmsInCore;
		CheckAlarm : FBCheckAlarmValues;
	END_VAR
END_FUNCTION_BLOCK
```

#### Types.typ - Exported data types
```iecst
(*----------------------------------------------------------------AlarmList------------------------------------------------------------------------------------------------------------------------------------------
В случае замены типов необходимо определить AlarmsListTypeSize*)

TYPE
	AlarmControlStatusTypeEnum :
		(
		AlarmControl_INIT := 0,
		AlarmControl_BIZY := 1,
		AlarmControl_DONE := 2,
		AlarmControl_ERROR := 3
		);
	AlarmBVMItemType : 	STRUCT  (*Alarm list boolean value monitor type*)
		Config : MpAlarmXAlarmConfigType; (*Alarm config*)
		Name : STRING[80]; (*Alarm name*)
		MonitoredValueAdr : UDINT; (*Adress of boolean monitored value*)
		TriggerValue : BOOL := TRUE;
	END_STRUCT;
END_TYPE
```

#### Constants.var - Exported constants
```iecst
VAR CONSTANT
	AlarmDVMListItemTypeSize : UINT := 892;
	AlarmDVMListItemTypeConfigSize : UINT := 800;
	AlarmDVMListItemTypeNameSize : UINT := 84;
	AlarmDVMListItemTypeMonValSize : UINT := 4;
	AlarmDVMListItemTypeTrigValSize : UINT := 1;
END_VAR
```

#### FBRecordAlarmsInCore.st
```iecst
(* TODO:  Done?*)
FUNCTION_BLOCK FBRecordAlarmsInCore
	CASE Status OF
		AlarmControl_INIT:
			IF Enable THEN
				MpAlarmXConfigAlarm_0.MpLink := ADR(AlarmXCore);
				MpAlarmXConfigAlarm_0.Enable := TRUE;
				MpAlarmXConfigAlarm_0.Configuration := ADR(MpAlarmXAlarmConfigType_0);
				Status := AlarmControl_BIZY;
				IF (Prefix <> '') THEN
					FOR i := 0 TO ListSize-1 DO
						AlarmBVMListItem ACCESS (AlarmBVMListAdr + AlarmDVMListItemTypeSize*i);
						// Добавление префикса к сообщению аларма
						AlarmBVMListItem.Config.Message := CONCAT(Prefix, AlarmBVMListItem.Config.Message);
					END_FOR
				END_IF

				IF (DeviceName <> '') THEN
					FOR i := 0 TO ListSize-1 DO
						AlarmBVMListItem ACCESS (AlarmBVMListAdr + AlarmDVMListItemTypeSize*i);
						// добавление имени устройства к имени аларма
						AlarmBVMListItem.Name := CONCAT(DeviceName, AlarmBVMListItem.Name);
					END_FOR
				END_IF
				i := 0;
			END_IF
		AlarmControl_BIZY:
			// производится запись ошибок из листа в ядро
			IF (i <= (ListSize-1)) THEN
				AlarmBVMListItem ACCESS (AlarmBVMListAdr + AlarmDVMListItemTypeSize*i);
				MpAlarmXConfigAlarm_0.Save := TRUE;
				MpAlarmXConfigAlarm_0.Name := ADR(AlarmBVMListItem.Name);
				MpAlarmXAlarmConfigType_0 := AlarmBVMListItem.Config;
				MpAlarmXConfigAlarm_0();
				IF ((MpAlarmXConfigAlarm_0.CommandDone) AND (NOT(MpAlarmXConfigAlarm_0.CommandBusy))) THEN
					i := i + 1;
					MpAlarmXConfigAlarm_0.Save := FALSE;
					MpAlarmXConfigAlarm_0();
				END_IF
				IF MpAlarmXConfigAlarm_0.Error THEN
					Status := AlarmControl_ERROR;
				END_IF
			ELSE
				Status := AlarmControl_DONE;
			END_IF
		AlarmControl_DONE:
			// Ошибки записаны, блок в режиме ожидания перезаписи
			IF NOT Enable THEN
				Status := AlarmControl_INIT;
			END_IF
		AlarmControl_ERROR:
			IF ResetError THEN
				IF MpAlarmXConfigAlarm_0.Error THEN
					MpAlarmXConfigAlarm_0.ErrorReset := TRUE;
					MpAlarmXConfigAlarm_0();
				ELSE
					ResetError := FALSE;
					Status := AlarmControl_INIT;
				END_IF
			END_IF
	END_CASE
END_FUNCTION_BLOCK
```

#### FBCheckAlarmValues.st
```iecst
(* TODO: Done?*)
FUNCTION_BLOCK FBCheckAlarmValues
	CASE Status OF
		AlarmControl_INIT:
			IF (AlarmBVMListAdr > 0) THEN
				IF Enable THEN
			(*	AlarmXCore ACCESS AlarmXCore;*)
				Status := AlarmControl_BIZY;
				END_IF
			ELSE
				Status := AlarmControl_ERROR;
				// AlarmBVMListAdr empty
			END_IF

		AlarmControl_BIZY:
			// Мониторинг переменных
			FOR i:=0 TO ListSize-1 DO
				AlarmListItem ACCESS (AlarmBVMListAdr + i*AlarmDVMListItemTypeSize);
				boolVal ACCESS (AlarmListItem.MonitoredValueAdr);
				IF (AlarmListItem.TriggerValue = boolVal) THEN
					AlarmXSetStatus := MpAlarmXSet(AlarmXCore, AlarmListItem.Name);
				ELSE
					AlarmXResetStatus := MpAlarmXReset(AlarmXCore, AlarmListItem.Name);
				END_IF
			END_FOR
			IF NOT Enable THEN
				Status := AlarmControl_DONE;
			END_IF
			// в случае возникновения ошибок Set/Reset алармов в ядре
//			IF ((AlarmXResetStatus <> 0) OR (AlarmXSetStatus <> 0)) THEN
//				Status := AlarmControl_ERROR;
//			END_IF

		AlarmControl_DONE:
			// Ожидание продолжения мониторинга переменных
			IF Enable THEN
				Status := AlarmControl_BIZY;
			END_IF;

		AlarmControl_ERROR:
			IF ResetError THEN
				Status := AlarmControl_INIT;
				ResetError := FALSE;
			END_IF
	END_CASE
END_FUNCTION_BLOCK
```

#### FBAlarmListControl.st
```iecst
(* TODO:  Done?*)
FUNCTION_BLOCK FBAlarmListControl
	CASE Status OF
		AlarmControl_INIT:
			RecordAlarm.AlarmBVMListAdr := AlarmBVMListAdr;
			RecordAlarm.AlarmXCore := AlarmXCore;
			RecordAlarm.ListSize := ListSize;
			RecordAlarm.Prefix := Prefix;
			RecordAlarm.DeviceName := DeviceName;
			RecordAlarm.Enable := TRUE;
			RecordAlarm();

			CheckAlarm.AlarmBVMListAdr := AlarmBVMListAdr;
			CheckAlarm.AlarmXCore := AlarmXCore;
			CheckAlarm.ListSize := ListSize;
			CheckAlarm.Enable := TRUE;
			Status := AlarmControl_BIZY;
		AlarmControl_BIZY:
			// Ожидание записи Аларм листа в ядро
			RecordAlarm();
			IF (RecordAlarm.Status = AlarmControl_DONE) THEN
				Status := AlarmControl_DONE;
			END_IF
			IF  RecordAlarm.Status = AlarmControl_ERROR THEN
				Status := AlarmControl_ERROR;
			END_IF;
		AlarmControl_DONE:
			// Мониторинг переменных, основной режим работы функционального блока
			CheckAlarm();
			IF CheckAlarm.Status = AlarmControl_ERROR THEN
				Status := AlarmControl_ERROR;
			END_IF
			IF NOT Enable THEN
				RecordAlarm.Enable := FALSE;
				RecordAlarm();
				CheckAlarm.Enable := FALSE;
				CheckAlarm();
				Status := AlarmControl_INIT;
			END_IF
		AlarmControl_ERROR:
			// Сброс ошибок в подконтрольных фб
			IF ResetError THEN
				IF  RecordAlarm.Status = AlarmControl_ERROR THEN
					RecordAlarm.ResetError := TRUE;
					RecordAlarm();
				END_IF;
				IF CheckAlarm.Status = AlarmControl_ERROR THEN
					CheckAlarm.ResetError := TRUE;
					CheckAlarm();
				END_IF
				IF ((RecordAlarm.Status <> AlarmControl_ERROR) AND (CheckAlarm.Status <> AlarmControl_ERROR)) THEN
					Status := AlarmControl_INIT;
					ResetError := FALSE;
				END_IF
			END_IF
	END_CASE
END_FUNCTION_BLOCK
```

- Visualisation Logical/mappView (not shown)

### Program Logical/ReadData (IEC)

#### Main.st - Init, cyclic, exit code
```iecst
PROGRAM _INIT
	(* Insert code here *)
	Step := 1;
	i := 0;
	j := 0;
END_PROGRAM

PROGRAM _CYCLIC
	(* Insert code here *)
	IF Start THEN
		CASE Step OF
			0 : (*error*)
			1 : (*init*)
				i := 0;
				Step := 4;
				offset := 0;
				val := 0;
				flag := FALSE;
				FBRead.Enable := TRUE;
				FBRead.strDevice := 'HardDisk';
				FBRead.strFile := 'TestFile1';
			2 : (*parsing*)
				SeparatorPosition := FIND(buffer_str,',');
				WHILE SeparatorPosition > 0 DO
					//				IF SeparatorPosition > 0 THEN
					IF SeparatorPosition > 1 THEN
						temp_str := MID(buffer_str,SeparatorPosition - 1,1);
						NewLinePosition := FIND(temp_str,'$n');
						IF NewLinePosition > 0 THEN
							temp_str := DELETE(temp_str,NewLinePosition,1);
						END_IF
						buffer_str := DELETE(buffer_str,SeparatorPosition,1);
						ReadedValue := STRING_TO_REAL(temp_str);
						temp_str := '';
						CASE val OF
							1: W[i] := ReadedValue;
								val := val + 1;
							3: IF i=0 THEN
									Velocity := ReadedValue;
									IF flag THEN
										V[0] := V[2399] + Velocity/100000;
										T[0] := T[2399] + 0.001;
									ELSE
										V[0] := 0;
										T[0] := 0;
									END_IF
								ELSE
									V[i] := V[i-1] + Velocity/100000;
									T[i] := T[i-1] + 0.001;
								END_IF
								val := val + 1;
							7: val := 0;
								IF flag THEN
									Ktare[j] := FFeederRatio(ADR(W), ADR(V), ADR(T), 2400);
									IF flag1 THEN
										StdDeviation := FStdDeviation(ADR(Ktare),2400);
									ELSE
										StdDeviation := FStdDeviation(ADR(Ktare),j);
									END_IF
									Rate := Velocity*Ktare[j];
									IF j = 2399 THEN
										j := 0;
										flag1 := TRUE;
									ELSE
										j := j + 1;
									END_IF
								ELSE
									IF i > 200 THEN
										Ktare[j] := FFeederRatio(ADR(W), ADR(V), ADR(T), i+1);
										Rate := Velocity*Ktare[j];
										IF (j>10) THEN
											StdDeviation := FStdDeviation(ADR(Ktare),j);
										END_IF
										IF j = 2399 THEN
											j := 0;
										ELSE
											j := j + 1;
										END_IF
									END_IF
								END_IF

								IF i = 2399 THEN
									i := 0;
									flag := TRUE;
								ELSE
									i := i + 1;
								END_IF
							ELSE
								val := val + 1;
						END_CASE
					ELSE
						buffer_str := DELETE(buffer_str,1,1);
					END_IF
					//				ELSE
					SeparatorPosition := FIND(buffer_str,',');
				END_WHILE
				Step := 3;
				//				END_IF
			3 : (*end of buffer*)
				Step := 4;
				offset := offset + BytesToRead - LEN(buffer_str);
			4 : (*read file*)
				FBRead.Read := TRUE;
				FBRead.BytesToRead := BytesToRead;
				FBRead.Offset := offset;
				FBRead();
				IF (FBRead.wStatus = 0) AND (FBRead.byStep = 3) THEN
					Step := 5;
					buffer_str := FBRead.ReadedStr;
				END_IF
			5 : (*check end of line*)
				//				NewLinePosition := FIND(buffer_str,'$n');
				Step := 2;
			ELSE
				Step := 0;
		END_CASE
	END_IF
END_PROGRAM

PROGRAM _EXIT
				(* Insert code here *)

				END_PROGRAM
```

#### Variables.var - Local variables
```iecst
VAR
	Velocity : REAL;
	SeparatorPosition : INT;
	NewLinePosition : INT;
	buffer_str : STRING[255];
	BytesToRead : UDINT := 255; (*equal to length of buffer_str*)
	temp_str : STRING[80]; (*for value*)
	Step : USINT; (*step of program*)
	offset : UDINT;
	Start : BOOL; (*trigger*)
	ReadedValue : REAL;
	i : UDINT; (*index*)
	j : UDINT;
	val : USINT;
	flag1 : BOOL := FALSE;
	flag : BOOL;
	FBRead : FBReadFromFile;
	Rate : REAL;
	StdDeviation : REAL;
END_VAR
```

#### LocalFunctions.fun
```iecst
{REDUND_ERROR} {REDUND_UNREPLICABLE} FUNCTION_BLOCK FBReadFromFile (*TODO: Add your comment here*) (*$GROUP=User,$CAT=User,$GROUPICON=User.png,$CATICON=User.png*)
	VAR_INPUT
		Enable : {REDUND_UNREPLICABLE} BOOL;
		BytesToRead : {REDUND_UNREPLICABLE} UDINT;
		Offset : {REDUND_UNREPLICABLE} UDINT := 0;
		Read : {REDUND_UNREPLICABLE} BOOL;
		strDevice : {REDUND_UNREPLICABLE} STRING[80];
		strFile : {REDUND_UNREPLICABLE} STRING[80];
	END_VAR
	VAR_OUTPUT
		ReadedStr : {REDUND_UNREPLICABLE} STRING[255];
		bOK : {REDUND_UNREPLICABLE} BOOL := FALSE;
		byStep : {REDUND_UNREPLICABLE} USINT := 1;
		byErrorLevel : {REDUND_UNREPLICABLE} USINT := 0;
		dwIdent : {REDUND_UNREPLICABLE} UDINT;
		wStatus : {REDUND_UNREPLICABLE} UINT;
		wError : {REDUND_UNREPLICABLE} UINT;
	END_VAR
	VAR
		FOpen : {REDUND_UNREPLICABLE} FileOpen;
		FRead : {REDUND_UNREPLICABLE} FileRead;
		FClose : {REDUND_UNREPLICABLE} FileClose;
	END_VAR
END_FUNCTION_BLOCK
```

#### FBReadFromFile.st
```iecst
(* TODO: Add your comment here *)
FUNCTION_BLOCK FBReadFromFile
	CASE byStep OF
		0: (**** Error step ****)
			bOK := FALSE;
			byStep := 1;
		1: (**** Try to open existing file ****)
			(* Initialize file open structrue *)
			FOpen.enable    := 1;
			FOpen.pDevice   := ADR(strDevice);
			FOpen.pFile     := ADR(strFile);
			FOpen.mode      := fiREAD_ONLY;  (* Read and write access *)
			(* Call FBK *)
			FOpen();
			(* Get FBK output information *)
			dwIdent := FOpen.ident;
			wStatus := FOpen.status;
			(* Verify status (20708 -> File doesn't exist) *)
			IF (wStatus = 20708) THEN
				byStep := 0;
				//				ошибка нет файла
			ELSE
				byStep := 4;
				//				IF (wStatus = 0) THEN
				//					byStep := 3;
				//				ELSE
				//					IF (wStatus <> 65535) THEN
				//						byErrorLevel := 1;
				//						byStep := 0;
				//						IF (wStatus = 20799) THEN
				//							wError := FileIoGetSysError();
				//						END_IF
				//					END_IF
				//				END_IF
			END_IF
		2: (**** Wait for restart ****)
			IF Enable THEN
				byStep := 1;
			END_IF
			//		2: (**** Create file ****)
			//			(* Initialize file create structure *)
			//			FCreate.enable  := 1;
			//			FCreate.pDevice := ADR(strDevice);
			//			FCreate.pFile   := ADR(strFile);
			//			(* Call FBK *)
			//			FCreate();
			//			(* Get FBK output information *)
			//			dwIdent := FCreate.ident;
			//			wStatus := FCreate.status;
			//			(* Verify status *)
			//			IF (wStatus = 0) THEN
			//				byStep := 3;
			//			ELSE
			//				IF (wStatus <> 65535) THEN
			//					byErrorLevel := 2;
			//					byStep := 0;
			//					IF (wStatus = 20799) THEN
			//						wError := FileIoGetSysError();
			//					END_IF
			//				END_IF
			//			END_IF
		3: (**** Wait for command ****)
			IF Read THEN
				byStep := 4;
			END_IF
			//		3: (**** Write data to file ****)
			//			(* Initialize file write structure *)
			//			FWrite.enable   := 1;
			//			FWrite.ident    := dwIdent;
			//			FWrite.offset   := 0;
			//			FWrite.pSrc     := ADR(byWriteData[0]);
			//			FWrite.len      := SIZEOF(byWriteData);
			//			(* Call FBK *)
			//			FWrite();
			//			(* Get status *)
			//			wStatus := FWrite.status;
			//			(* Verify status *)
			//			IF (wStatus = 0) THEN
			//				byStep := 4;
			//			ELSE
			//				IF (wStatus <> 65535) THEN
			//					byErrorLevel := 3;
			//					byStep := 0;
			//					IF (wStatus = 20799) THEN
			//						wError := FileIoGetSysError();
			//					END_IF
			//				END_IF
			//			END_IF
		4: (**** Read data from file ****)
			(* Initialize file read structure *)
			FRead.enable    := 1;
			FRead.ident     := dwIdent;
			FRead.offset    := Offset;
			FRead.pDest     := ADR(ReadedStr);
			FRead.len       := BytesToRead;
			(* Call FBK *)
			IF Read THEN
				FRead();
				(* Get status *)
				wStatus := FRead.status;
				(* Verify status *)
				IF (wStatus = 0) THEN
					Read := FALSE;
					byStep := 3;
//					ReadedStr := DELETE(ReadedStr,10000,UDINT_TO_INT(BytesToRead+1));
				ELSE
					IF (wStatus <> 65535) THEN
						byErrorLevel := 4;
						byStep := 0;
						IF (wStatus = 20799) THEN
							wError := FileIoGetSysError();
						END_IF
					END_IF
				END_IF
			END_IF
		5: (**** Close file ****)
			(* Initialize file close structure *)
			FClose.enable   := 1;
			FClose.ident    := dwIdent;
			(* Call FBK *)
			FClose();
			(* Get status *)
			wStatus := FClose.status;
			(* Verify status *)
			IF (wStatus = 0) THEN
				Enable := FALSE;
				byStep := 2;
			ELSE
				IF (wStatus <> 65535) THEN
					byErrorLevel := 5;
					byStep := 0;
					IF (wStatus = 20799) THEN
						wError := FileIoGetSysError();
					END_IF
				END_IF
			END_IF
		//		6: (**** Delete file ****)
		//			(* Initialize file delete structure *)
		//			FDelete.enable  := 1;
		//			FDelete.pDevice := ADR(strDevice);
		//			FDelete.pName   := ADR(strFile);
		//			(* Call FBK *)
		//			FDelete();
		//			(* Get status *)
		//			wStatus := FDelete.status;
		//			(* Verify status *)
		//			IF (wStatus = 0) THEN
		//				bOK     := TRUE;
		//				byStep := 7;
		//			ELSE
		//				IF (wStatus <> 65535) THEN
		//					byErrorLevel := 6;
		//					byStep := 0;
		//					IF (wStatus = 20799) THEN
		//						wError := FileIoGetSysError();
		//					END_IF
		//				END_IF
		//			END_IF
	END_CASE
END_FUNCTION_BLOCK
```

### Data object Logical/acp10etxen (Ett)

- acp10etxen.ett (not shown)

### Package Logical/gAxis01obj - gAxis01obj

### gAxis01i.ax
```
InitParameter (Version=5.01.1, NcSwId=Acp10)
  ACP10AXIS_typ:
    dig_in:
      level:
        reference = ncACTIV_HI
        pos_hw_end = ncACTIV_LO
        neg_hw_end = ncACTIV_LO
        trigger1 = ncACTIV_HI
        trigger2 = ncACTIV_HI
    encoder_if:
      parameter:
        count_dir = ncSTANDARD
        scaling:
          load:
            units = 1000
            rev_motor = 1
    limit:
      parameter:
        v_pos = 10000
        v_neg = 0.0
        a1_pos = 50000
        a2_pos = 50000
        a1_neg = 50000
        a2_neg = 50000
        t_jolt = 0
        t_in_pos = 0
        pos_sw_end = 2000000000
        neg_sw_end = -2000000000
        ds_warning = 1000.0
        ds_stop = 1000
        a_stop = 1.0e30
        dv_stop = 0
        dv_stop_mode = ncOFF
    controller:
      mode = ncPOSITION
      position:
        kv = 50
        tn = 0
        t_predict = 0.0004
        t_total = 0.0004
        p_max = 1.0e30
        i_max = 0
      speed:
        kv = 0.2
        tn = 0
        t_filter = 0.0
        isq_filter1:
          type = ncOFF
          a0 = 0.0
          a1 = 0.0
          b0 = 0.0
          b1 = 0.0
          b2 = 0.0
          c0_par_id = 0
          c1_par_id = 0
        isq_filter2:
          type = ncOFF
          a0 = 0.0
          a1 = 0.0
          b0 = 0.0
          b1 = 0.0
          b2 = 0.0
          c0_par_id = 0
          c1_par_id = 0
        isq_filter3:
          type = ncOFF
          a0 = 0.0
          a1 = 0.0
          b0 = 0.0
          b1 = 0.0
          b2 = 0.0
          c0_par_id = 0
          c1_par_id = 0
      uf:
        type = ncLINEAR
        auto_config = ncMOTOR_PAR
        u0 = 0
        un = 0
        fn = 50.0
        k_f_slip = 0
      ff:
        torque_load = 0.0
        torque_pos = 0.0
        torque_neg = 0.0
        kv_torque = 0.0
        inertia = 0.0
        t_filter_a = 0.0
    move:
      stop:
        parameter[0]:
          decel_ramp = ncA_LIMIT
          controller = ncON
        parameter[1]:
          decel_ramp = ncA_LIMIT
          controller = ncON
        parameter[2]:
          decel_ramp = ncA_LIMIT
          controller = ncON
        parameter[3]:
          decel_ramp = ncA_LIMIT
          controller = ncON
        quickstop:
          decel_ramp = ncA_LIMIT
        drive_error:
          decel_ramp = ncA_LIMIT
      homing:
        parameter:
          s = 0
          v_switch = 5000
          v_trigger = 500
          a = 50000
          mode = ncDIRECT
          edge_sw = ncPOSITIVE
          start_dir = ncPOSITIVE
          trigg_dir = ncPOSITIVE
          ref_pulse = ncOFF
          fix_dir = ncOFF
          tr_s_block = 0
          torque_lim = 0
          ds_block = 0
          ds_stop = 0
      basis:
        parameter:
          v_pos = 10000.0
          v_neg = 0.0
          a1_pos = 50000
          a2_pos = 50000
          a1_neg = 50000
          a2_neg = 50000
    message:
      text:
        parameter:
          format = ncBREAK
          columns = 80
          data_modul = acp10etxen
```

### Program Logical/HWtest (IEC)

#### Variables.var
```iecst
VAR
	FeederBlock : FBFeederBlock;
	ConfigS : FeederConfigType;
	ConfigP : FeederConfigType;
	Par1 : MpAxisBasicParType := (Acceleration:=50000,Deceleration:=50000,Velocity:=10000);
	CyclicSet1 : MpAxisCyclicSetParType := (Acceleration:=50000,Deceleration:=50000,PositionModeMaxVelocity:=10000);
	Par2 : MpAxisBasicParType := (Acceleration:=50000,Deceleration:=50000,Velocity:=10000);
	CyclicSet2 : MpAxisCyclicSetParType := (Acceleration:=50000,Deceleration:=50000,PositionModeMaxVelocity:=10000);
	FeederConfig : FeederBlockConfigType;
	MpAlarmXCore_0 : MpAlarmXCore; (*MpRecipeXml_0 : MpRecipeXml;
	MpRecipeRegPar_0 : MpRecipeRegPar;*)
	Counter : FBSpendTotalizer;
	var : REAL;
	Control : FeederBlockControlType;
END_VAR
```

#### Main.st
```iecst
PROGRAM _INIT
	(* Insert code here *)

	Config.AlarmPrefix := '123123';

	Config.WarningWeight := 0.3;
	Config.AlarmWeight := 0.1;
	Config.ResetWeightLimit := 0.1;

	Config.DefaultTareK := 0.85;
	Config.DeviationLimit := 0.1;
	Config.EnableAutoRateControl := FALSE;

	Config.TareCalcDelay := T#10s;
	Config.ToGoToAutoDelay := T#10s;
	Config.BufferDelay := T#10s;
	Config.DeviationCalcDelay := T#10s;

	Config.Handler.ACPConfigLink := ADR(gAxis01);
	Config.Handler.AxisBasicParLink := ADR(Par1);
	Config.Handler.AxisConfigLink := ADR(gLinkFeeder1);
	Config.Handler.AxisCyclicSetParLink := ADR(CyclicSet1);
	Config.Handler.PostpurgeTime := T#5s;
	Config.Handler.PrepurgeTime := T#5s;
	Config.Handler.GasCalibrateOut.A :=  -0.12890000641345978;
	Config.Handler.GasCalibrateOut.B := 659.57000732421875;
	Config.Handler.GasCalibrateOut.C := 105.16000366210938;
	Config.Handler.GasCalibrateOut.MaxValue := 9969;
	Config.Handler.GasCalibrateOut.MinValue := 0;

	Config.WeightCalibrate.A := 0;
	Config.WeightCalibrate.B := 5.82e-05;
	Config.WeightCalibrate.C := -5.4242;
	Config.WeightCalibrate.MaxValue := 60;
	Config.WeightCalibrate.MinValue := 0;

	Config.GasCalibrateIn.A := 0;
	Config.GasCalibrateIn.B := 0.0038000000640749931;
	Config.GasCalibrateIn.C := -12.600000381469727;
	Config.GasCalibrateIn.MaxValue := 50;
	Config.GasCalibrateIn.MinValue := 0;

	FeederBlock.Config.PrimaryFeeder := Config;
	Config.Handler.ACPConfigLink := ADR(gAxis02);
	Config.Handler.AxisBasicParLink := ADR(Par2);
	Config.Handler.AxisConfigLink := ADR(gLinkFeeder2);
	Config.Handler.AxisCyclicSetParLink := ADR(CyclicSet2);
	Config.WeightCalibrate.C := -5.2;
	FeederBlock.Config.SecondaryFeeder := Config;

	FeederBlock.Control.PrimaryFeeder.Handler.KZP := 100;
	FeederBlock.Control.PrimaryFeeder.Handler.KZU := 0;
	//	Handler.Config := Config.Handler;
	FeederBlock.Config.DualFeederMode := TRUE;
	FeederBlock.Enable := TRUE;
END_PROGRAM

PROGRAM _CYCLIC
	(* Insert code here *)
	FeederBlock();
//	Handler();
END_PROGRAM

PROGRAM _EXIT
	(* Insert code here *)

END_PROGRAM
```

### Library Logical/FeederLib (IEC, version 1.00.4)
Depends on: MpAxis, Acp10_MC, NcGlobal, MpBase, MpCom, brsystem, Acp10man, Acp10par, UserLib, UsAlarmLib

#### Types.typ - Exported data types
```iecst
(*FBFeederHandler*)

TYPE
	FeederHandlerStatusEnum :
		(
		FEEDCTRL_ERROR := 0,
		FEEDCTRL_INIT := 1,
		FEEDCTRL_READY_TO_FEED := 2,
		FEEDCTRL_PREPURGE := 3,
		FEEDCTRL_FEEDING := 4,
		FEEDCTRL_POSTPURGE := 5
		);
	FeederHandlerControlType : 	STRUCT
		PowderRate : UINT; (*Базовое управляющее значение расхода порошка*)
		KZP : REAL;
		KZU : REAL;
		GasRate : UINT; (*Управляющее значение расходом газа*)
	END_STRUCT;
	FeederHandlerConfigType : 	STRUCT
		PrepurgeTime : TIME;
		PostpurgeTime : TIME;
		AxisConfigLink : UDINT;
		ACPConfigLink : UDINT;
		AxisBasicParLink : UDINT;
		AxisCyclicSetParLink : UDINT;
		GasCalibrateOut : CalibrationType;
		Ratio : USINT := 25;
	END_STRUCT;
	FeederHandlerIOoutType : 	STRUCT
		aoGasRate : INT; (*Управление регулятором расхода*)
		doShutOff : BOOL;
		doMixer : BOOL;
	END_STRUCT;
	FeederHandlerIOinType : 	STRUCT
		aiGasRate : UINT; (*Показание регулятора расхода*)
	END_STRUCT;
	FeederHandlerUserInfoType : 	STRUCT
		Active : BOOL;
		ActualSpeed : REAL;
	END_STRUCT;
	FeederHandlerIOType : 	STRUCT
		In : FeederHandlerIOinType;
		Out : FeederHandlerIOoutType;
	END_STRUCT;
END_TYPE

(*FBFeeder*)

TYPE
	FeederStatusEnum :
		(
		FEED_ERROR := 0,
		FEED_INIT := 1,
		FEED_PAUSE := 2,
		FEED_RESET := 3,
		FEED_READY := 4,
		FEED_FEEDING := 5
		);
	FeederControlType : 	STRUCT
		Handler : FeederHandlerControlType;
		ManualTareControl : BOOL;
		TareK : REAL;
	END_STRUCT;
	FeederConfigType : 	STRUCT
		Handler : FeederHandlerConfigType;
		GasCalibrateIn : CalibrationType;
		WeightCalibrate : CalibrationType;
		DefaultTareK : REAL;
		WarningWeight : REAL;
		AlarmWeight : REAL;
		AlarmPrefix : STRING[80];
		EnableAutoRateControl : BOOL;
		BufferDelay : TIME;
		TareCalcDelay : TIME;
		DeviationCalcDelay : TIME;
		ToGoToAutoDelay : TIME;
		RecordInBufferPerion : TIME := T#100ms; (*Запись значений в буфер через указанное время*)
		DeviationLimit : REAL;
		ResetWeightLimit : REAL;
		ControlWord : UINT := 29828;
	END_STRUCT;
	FeederIOinType : 	STRUCT
		Handler : FeederHandlerIOinType;
		aiWeight : DINT;
	END_STRUCT;
	FeederUserInfoType : 	STRUCT
		Handler : FeederHandlerUserInfoType;
		Weight : REAL;
		Rate : REAL;
		TareK : REAL;
		Deviation : REAL;
		IsAUTO : BOOL;
	END_STRUCT;
END_TYPE

(*FBFeederBlock*)

TYPE
	FeederBlockStatusEnum :
		(
		FEEDBLOCK_ERROR := 0,
		FEEDBLOCK_INIT := 1,
		FEEDBLOCK_SINGLE := 2,
		FEEDBLOCK_DUAL := 3
		);
	FeederBlockControlType : 	STRUCT
		PrimaryFeeder : FeederControlType;
		SecondaryFeeder : FeederControlType;
		PrimaryStart : BOOL;
		SecondaryStart : BOOL;
		SeparateMode : BOOL;
		FeederSwitch : BOOL;
	END_STRUCT;
	FeederBlockConfigType : 	STRUCT
		PrimaryFeeder : FeederConfigType;
		SecondaryFeeder : FeederConfigType;
		DualFeederMode : BOOL;
	END_STRUCT;
	FeederBlockIOinType : 	STRUCT
		PrimaryFeeder : FeederIOinType;
		SecondaryFeeder : FeederIOinType;
	END_STRUCT;
	FeederBlockIOoutType : 	STRUCT
		PrimaryFeeder : FeederHandlerIOoutType;
		SecondaryFeeder : FeederHandlerIOoutType;
	END_STRUCT;
	FeederBlockUserInfoType : 	STRUCT
		PrimaryFeeder : FeederUserInfoType;
		SecondaryFeeder : FeederUserInfoType;
	END_STRUCT;
END_TYPE
```

#### FeederLib.fun - Exported functions and function blocks
```iecst
(*Insert your comment here.*)

{REDUND_ERROR} FUNCTION FFeederRatio : REAL (*TODO: Add your comment here*) (*$GROUP=User,$CAT=User,$GROUPICON=User.png,$CATICON=User.png*)
	VAR_INPUT
		W : REFERENCE TO ARRAY[0..2399] OF REAL;
		V : REFERENCE TO ARRAY[0..2399] OF REAL;
		T : REFERENCE TO ARRAY[0..2399] OF REAL;
		lengthOfArray : UDINT;
	END_VAR
	VAR
		sxx : LREAL;
		sxy : LREAL;
		sxp : LREAL;
		sumx : LREAL;
		sumy : LREAL;
		sump : LREAL;
		sumx2 : LREAL;
		sumxy : LREAL;
		sumxp : LREAL;
		i : UDINT;
	END_VAR
END_FUNCTION

{REDUND_ERROR} FUNCTION FStdDeviation : REAL (*TODO: Add your comment here*) (*$GROUP=User,$CAT=User,$GROUPICON=User.png,$CATICON=User.png*)
	VAR_INPUT
		Array : REFERENCE TO ARRAY[0..2399] OF REAL;
		lengthOfArray : UDINT;
	END_VAR
	VAR
		avg : REAL;
		sum : REAL;
		i : UDINT;
	END_VAR
END_FUNCTION

{REDUND_ERROR} FUNCTION_BLOCK FBFeederHandler (*TODO: Add your comment here*) (*$GROUP=User,$CAT=User,$GROUPICON=User.png,$CATICON=User.png*)
	VAR_INPUT
		Enable : BOOL;
		Start : BOOL;
		Config : FeederHandlerConfigType;
		Control : FeederHandlerControlType;
		TareK : REAL;
		IOin : FeederHandlerIOinType;
	END_VAR
	VAR_OUTPUT
		UserInfo : FeederHandlerUserInfoType;
		Status : FeederHandlerStatusEnum := FEEDCTRL_INIT;
		IOout : FeederHandlerIOoutType;
	END_VAR
	VAR
		AxisBasic : MpAxisBasic;
		AxisCyclicSet : MpAxisCyclicSet;
		TON_Prepurge : TON;
		TON_Postpurge : TON;
	END_VAR
END_FUNCTION_BLOCK

{REDUND_ERROR} FUNCTION_BLOCK FBFeeder (*TODO: Add your comment here*) (*$GROUP=User,$CAT=User,$GROUPICON=User.png,$CATICON=User.png*)
	VAR_INPUT
		Enable : {REDUND_UNREPLICABLE} BOOL;
		Reset : BOOL;
		Start : BOOL;
		Config : FeederConfigType;
		Control : FeederControlType;
		IOin : FeederIOinType;
	END_VAR
	VAR_OUTPUT
		IOout : FeederHandlerIOoutType;
		UserInfo : FeederUserInfoType;
		Status : FeederStatusEnum := FEED_INIT;
	END_VAR
	VAR
		FBControl : FBFeederHandler;
		TON_TareCalcDelay : TON;
		TON_DeviationCalcDelay : TON;
		TON_ToGoToAutoDelay : TON;
		TON_BufferDelay : TON;
		TON_WriteInBufferPeriod : TON := (PT:=T#100ms);
		WBuffer : ARRAY[0..2399] OF REAL;
		TBuffer : ARRAY[0..2399] OF REAL;
		PBuffer : ARRAY[0..2399] OF REAL;
		TareKBuffer : ARRAY[0..2399] OF REAL;
		i : UINT;
		j : UINT;
		WriteInWTP : BOOL := FALSE;
		WriteInTareK : BOOL := FALSE;
		RewriteWTP : BOOL := FALSE;
		RewriteTareK : BOOL := FALSE;
		CalcDeviation : BOOL := FALSE;
	END_VAR
END_FUNCTION_BLOCK

{REDUND_ERROR} FUNCTION_BLOCK FBFeederBlock (*TODO: Add your comment here*) (*$GROUP=User,$CAT=User,$GROUPICON=User.png,$CATICON=User.png*)
	VAR_INPUT
		Enable : {REDUND_UNREPLICABLE} BOOL;
		Control : FeederBlockControlType;
		Config : FeederBlockConfigType;
		IOin : FeederBlockIOinType;
	END_VAR
	VAR_OUTPUT
		Status : FeederBlockStatusEnum := FEEDBLOCK_INIT;
		IOout : FeederBlockIOoutType;
		UserInfo : FeederBlockUserInfoType;
	END_VAR
	VAR
		PrimaryFeeder : FBFeeder;
		SecondaryFeeder : FBFeeder;
	END_VAR
END_FUNCTION_BLOCK
```

#### FFeederRatio.st
```iecst
(* TODO: Add your comment here *)
FUNCTION FFeederRatio
	sumx := 0;
	sumy := 0;
	sump := 0;
	sumx2 := 0;
	sumxy := 0;
	sumxp := 0;

	FOR i := 0 TO lengthOfArray-1 DO
		sumy := sumy + W[i];
		sump := sump + V[i];
		sumx := sumx + T[i];
		sumx2 := sumx2 + T[i]*T[i];
		sumxy := sumxy + (W[i])*(T[i]);
		sumxp := sumxp + (V[i])*(T[i]);
	END_FOR

	sxx := sumx2 - (sumx*sumx)/UDINT_TO_LREAL(lengthOfArray);
	sxy := sumxy - (sumx*sumy)/UDINT_TO_LREAL(lengthOfArray);
	sxp := sumxp - (sumx*sump)/UDINT_TO_LREAL(lengthOfArray);

	FFeederRatio := LREAL_TO_REAL(-(sxy/sxx)/(sxp/sxx))*6;
END_FUNCTION
```

#### FStdDeviation.st
```iecst
(* TODO: Add your comment here *)
FUNCTION FStdDeviation
	sum := 0;
	FOR i := 0 TO lengthOfArray-1 DO
		sum := sum + Array[i];
	END_FOR
	avg := sum/lengthOfArray;
	sum := 0;
	FOR i := 0 TO lengthOfArray-1 DO
		sum := sum + EXPT(Array[i]-avg, 2);
	END_FOR
	FStdDeviation := SQRT(sum/lengthOfArray);
END_FUNCTION
```

#### FBFeederBlock.st
```iecst
(* TODO: Add your comment here *)
FUNCTION_BLOCK FBFeederBlock
	IF Enable THEN
		CASE Status OF
			FEEDBLOCK_ERROR:
			FEEDBLOCK_INIT:
				PrimaryFeeder.Config := Config.PrimaryFeeder;
				PrimaryFeeder.IOin := IOin.PrimaryFeeder;
				PrimaryFeeder.Enable := TRUE;
				IF Config.DualFeederMode THEN
					SecondaryFeeder.Config := Config.SecondaryFeeder;
					SecondaryFeeder.IOin := IOin.SecondaryFeeder;
					SecondaryFeeder.Enable := TRUE;
					PrimaryFeeder();
					SecondaryFeeder();
					IF (PrimaryFeeder.Status = FEED_READY) AND (SecondaryFeeder.Status = FEED_READY) THEN
						Status := FEEDBLOCK_DUAL;
					END_IF
				ELSE
					PrimaryFeeder();
					IF (PrimaryFeeder.Status = FEED_READY) THEN
						Status := FEEDBLOCK_SINGLE;
					END_IF
				END_IF
			FEEDBLOCK_SINGLE:
				PrimaryFeeder.Control := Control.PrimaryFeeder;
				PrimaryFeeder.IOin := IOin.PrimaryFeeder;
				PrimaryFeeder.Start := Control.PrimaryStart;
				PrimaryFeeder();
				IOout.PrimaryFeeder := PrimaryFeeder.IOout;
				UserInfo.PrimaryFeeder := PrimaryFeeder.UserInfo;
			FEEDBLOCK_DUAL:
				PrimaryFeeder.IOin := IOin.PrimaryFeeder;
				SecondaryFeeder.IOin := IOin.SecondaryFeeder;
				IF Control.SeparateMode THEN
					PrimaryFeeder.Control := Control.PrimaryFeeder;
					PrimaryFeeder.Start := Control.PrimaryStart;

					SecondaryFeeder.Control := Control.SecondaryFeeder;
					SecondaryFeeder.Start := Control.SecondaryStart;
				ELSE
					IF Control.FeederSwitch THEN
						SecondaryFeeder.Control := Control.PrimaryFeeder;
						SecondaryFeeder.Start := Control.PrimaryStart;
					ELSE
						PrimaryFeeder.Control := Control.PrimaryFeeder;
						PrimaryFeeder.Start := Control.PrimaryStart;
					END_IF
				END_IF
				PrimaryFeeder();
				SecondaryFeeder();

				IOout.PrimaryFeeder := PrimaryFeeder.IOout;
				UserInfo.PrimaryFeeder := PrimaryFeeder.UserInfo;

				IOout.SecondaryFeeder := SecondaryFeeder.IOout;
				UserInfo.SecondaryFeeder := SecondaryFeeder.UserInfo;
		END_CASE
	END_IF
END_FUNCTION_BLOCK
```
